LIN {X 0,Y 673.595,Z 978.183,A -85,B 0,C 180,E1 32397.712,E2 32397.712} C_VEL
LIN {X 0,Y 673.691,Z 963.128,A -85,B 0,C 180,E1 32397.38,E2 32397.38} C_VEL
LIN {X 0,Y 673.783,Z 926.963,A -85,B 0,C 180,E1 32396.96,E2 32396.96} C_VEL
LIN {X 0,Y 674.022,Z 820.76,A -85,B 0,C 180,E1 32395.779,E2 32395.779} C_VEL
LIN {X 0,Y 674.488,Z 777.084,A -85,B 0,C 180,E1 32392.62,E2 32392.62} C_VEL
LIN {X 0,Y 674.751,Z 739.413,A -85,B 0,C 180,E1 32389.928,E2 32389.928} C_VEL
LIN {X 0,Y 674.996,Z 702.216,A -85,B 0,C 180,E1 32387.302,E2 32387.302} C_VEL
LIN {X 0,Y 674.853,Z 660.758,A -85,B 0,C 180,E1 32384.443,E2 32384.443} C_VEL
LIN {X 0,Y 674.656,Z 625.3,A -85,B 0,C 180,E1 32382.074,E2 32382.074} C_VEL
LIN {X 0,Y 672.585,Z 616.892,A -85,B 0,C 180,E1 32381.448,E2 32381.448} C_VEL
LIN {X 0,Y 672.585,Z 616.892,A -85,B 0,C 180,E1 32378.297,E2 32378.297} C_VEL
LIN {X 0,Y 672.544,Z 616.896,A -85,B 0,C 180,E1 32375.211,E2 32375.211} C_VEL
LIN {X 0,Y 672.55,Z 616.893,A -85,B 0,C 180,E1 32372.362,E2 32372.362} C_VEL
LIN {X 0,Y 672.577,Z 616.89,A -85,B 0,C 180,E1 32369.233,E2 32369.233} C_VEL
LIN {X 0,Y 672.572,Z 616.892,A -85,B 0,C 180,E1 32366.203,E2 32366.203} C_VEL
LIN {X 0,Y 672.574,Z 616.893,A -85,B 0,C 180,E1 32363.191,E2 32363.191} C_VEL
LIN {X 0,Y 672.566,Z 616.892,A -85,B 0,C 180,E1 32360.227,E2 32360.227} C_VEL
LIN {X 0,Y 672.576,Z 616.888,A -85,B 0,C 180,E1 32357.086,E2 32357.086} C_VEL
LIN {X 0,Y 672.546,Z 616.892,A -85,B 0,C 180,E1 32354.087,E2 32354.087} C_VEL
LIN {X 0,Y 672.591,Z 616.89,A -85,B 0,C 180,E1 32351.076,E2 32351.076} C_VEL
LIN {X 0,Y 672.582,Z 616.891,A -85,B 0,C 180,E1 32347.984,E2 32347.984} C_VEL
LIN {X 0,Y 672.581,Z 616.892,A -85,B 0,C 180,E1 32344.851,E2 32344.851} C_VEL
LIN {X 0,Y 672.566,Z 616.895,A -85,B 0,C 180,E1 32344.293,E2 32344.293} C_VEL
LIN {X 0,Y 678.826,Z 637.109,A -85,B 0,C 180,E1 32342.275,E2 32342.275} C_VEL
LIN {X 0,Y 677.864,Z 671.07,A -85,B 0,C 180,E1 32339.563,E2 32339.563} C_VEL
LIN {X 0,Y 677.664,Z 682.912,A -85,B 0,C 180,E1 32338.655,E2 32338.655} C_VEL
LIN {X 0,Y 681.031,Z 699.716,A -85,B 0,C 180,E1 32338.3,E2 32338.3} C_VEL
LIN {X 0,Y 679.199,Z 978.779,A -85,B 0,C 180,E1 32335.156,E2 32335.156} C_VEL
LIN {X 0,Y 678.886,Z 1000.715,A -85,B 0,C 180,E1 32334.812,E2 32334.812} C_VEL
LIN {X 0,Y 678.362,Z 1022.472,A -85,B 0,C 180,E1 32334.307,E2 32334.307} C_VEL
LIN {X 0,Y 677.771,Z 1043.763,A -85,B 0,C 180,E1 32333.656,E2 32333.656} C_VEL
LIN {X 0,Y 677.123,Z 1063.834,A -85,B 0,C 180,E1 32332.892,E2 32332.892} C_VEL
LIN {X 0,Y 676.435,Z 1082.877,A -85,B 0,C 180,E1 32332.005,E2 32332.005} C_VEL
LIN {X 0,Y 675.676,Z 1102.121,A -85,B 0,C 180,E1 32330.942,E2 32330.942} C_VEL
LIN {X 0,Y 674.981,Z 1120.021,A -85,B 0,C 180,E1 32329.783,E2 32329.783} C_VEL
LIN {X 0,Y 674.308,Z 1136.916,A -85,B 0,C 180,E1 32328.5,E2 32328.5} C_VEL
LIN {X 0,Y 673.686,Z 1152.877,A -85,B 0,C 180,E1 32327.088,E2 32327.088} C_VEL
LIN {X 0,Y 673.175,Z 1167.476,A -85,B 0,C 180,E1 32325.594,E2 32325.594} C_VEL
LIN {X 0,Y 672.763,Z 1180.671,A -85,B 0,C 180,E1 32324.018,E2 32324.018} C_VEL
LIN {X 0,Y 672.436,Z 1192.394,A -85,B 0,C 180,E1 32322.363,E2 32322.363} C_VEL
LIN {X 0,Y 672.2,Z 1203.223,A -85,B 0,C 180,E1 32320.541,E2 32320.541} C_VEL
LIN {X 0,Y 672.056,Z 1211.703,A -85,B 0,C 180,E1 32318.814,E2 32318.814} C_VEL
LIN {X 0,Y 671.961,Z 1218.677,A -85,B 0,C 180,E1 32317.007,E2 32317.007} C_VEL
LIN {X 0,Y 671.917,Z 1224.198,A -85,B 0,C 180,E1 32315.121,E2 32315.121} C_VEL
LIN {X 0,Y 671.906,Z 1227.88,A -85,B 0,C 180,E1 32313.326,E2 32313.326} C_VEL
LIN {X 0,Y 671.901,Z 1229.885,A -85,B 0,C 180,E1 32311.534,E2 32311.534} C_VEL
LIN {X 0,Y 671.899,Z 1230.396,A -85,B 0,C 180,E1 32309.573,E2 32309.573} C_VEL
LIN {X 0,Y 671.913,Z 1229.232,A -85,B 0,C 180,E1 32307.696,E2 32307.696} C_VEL
LIN {X 0,Y 671.922,Z 1226.459,A -85,B 0,C 180,E1 32305.903,E2 32305.903} C_VEL
LIN {X 0,Y 671.934,Z 1221.905,A -85,B 0,C 180,E1 32304.02,E2 32304.02} C_VEL
LIN {X 0,Y 671.99,Z 1215.93,A -85,B 0,C 180,E1 32302.217,E2 32302.217} C_VEL
LIN {X 0,Y 672.093,Z 1208.469,A -85,B 0,C 180,E1 32300.494,E2 32300.494} C_VEL
LIN {X 0,Y 672.279,Z 1198.83,A -85,B 0,C 180,E1 32298.677,E2 32298.677} C_VEL
LIN {X 0,Y 672.551,Z 1188.342,A -85,B 0,C 180,E1 32297.026,E2 32297.026} C_VEL
LIN {X 0,Y 672.903,Z 1175.746,A -85,B 0,C 180,E1 32295.367,E2 32295.367} C_VEL
LIN {X 0,Y 673.372,Z 1161.698,A -85,B 0,C 180,E1 32293.789,E2 32293.789} C_VEL
LIN {X 0,Y 673.953,Z 1146.187,A -85,B 0,C 180,E1 32292.293,E2 32292.293} C_VEL
LIN {X 0,Y 674.602,Z 1129.671,A -85,B 0,C 180,E1 32290.923,E2 32290.923} C_VEL
LIN {X 0,Y 675.282,Z 1112.074,A -85,B 0,C 180,E1 32289.682,E2 32289.682} C_VEL
LIN {X 0,Y 676.046,Z 1092.906,A -85,B 0,C 180,E1 32288.526,E2 32288.526} C_VEL
LIN {X 0,Y 676.778,Z 1073.721,A -85,B 0,C 180,E1 32287.547,E2 32287.547} C_VEL
LIN {X 0,Y 677.469,Z 1053.6,A -85,B 0,C 180,E1 32286.699,E2 32286.699} C_VEL
LIN {X 0,Y 678.09,Z 1032.642,A -85,B 0,C 180,E1 32285.984,E2 32285.984} C_VEL
LIN {X 0,Y 678.646,Z 1011.301,A -85,B 0,C 180,E1 32285.414,E2 32285.414} C_VEL
LIN {X 0,Y 679.058,Z 989.931,A -85,B 0,C 180,E1 32285,E2 32285} C_VEL
LIN {X 0,Y 679.387,Z 956.893,A -85,B 0,C 180,E1 32284.593,E2 32284.593} C_VEL
LIN {X 0,Y 680.928,Z 698.596,A -85,B 0,C 180,E1 32281.704,E2 32281.704} C_VEL
LIN {X 0,Y 677.358,Z 681.383,A -85,B 0,C 180,E1 32281.33,E2 32281.33} C_VEL
LIN {X 0,Y 678.154,Z 642.731,A -85,B 0,C 180,E1 32278.338,E2 32278.338} C_VEL
LIN {X 0,Y 678.247,Z 636.016,A -85,B 0,C 180,E1 32277.803,E2 32277.803} C_VEL
LIN {X 0,Y 672.566,Z 616.894,A -85,B 0,C 180,E1 32275.91,E2 32275.91} C_VEL
LIN {X 0,Y 672.583,Z 616.889,A -85,B 0,C 180,E1 32272.831,E2 32272.831} C_VEL
LIN {X 0,Y 672.559,Z 616.894,A -85,B 0,C 180,E1 32269.817,E2 32269.817} C_VEL
LIN {X 0,Y 672.579,Z 616.886,A -85,B 0,C 180,E1 32266.853,E2 32266.853} C_VEL
LIN {X 0,Y 672.553,Z 616.894,A -85,B 0,C 180,E1 32263.735,E2 32263.735} C_VEL
LIN {X 0,Y 672.566,Z 616.888,A -85,B 0,C 180,E1 32260.824,E2 32260.824} C_VEL
LIN {X 0,Y 672.548,Z 616.894,A -85,B 0,C 180,E1 32257.666,E2 32257.666} C_VEL
LIN {X 0,Y 672.546,Z 616.891,A -85,B 0,C 180,E1 32254.814,E2 32254.814} C_VEL
LIN {X 0,Y 672.548,Z 616.896,A -85,B 0,C 180,E1 32251.657,E2 32251.657} C_VEL
LIN {X 0,Y 672.584,Z 617.001,A -85,B 0,C 180,E1 32249.822,E2 32249.822} C_VEL
LIN {X 0,Y 675.411,Z 626.556,A -85,B 0,C 180,E1 32248.699,E2 32248.699} C_VEL
LIN {X 0,Y 680.163,Z 637.227,A -85,B 0,C 180,E1 32248.344,E2 32248.344} C_VEL
LIN {X 0,Y 681.085,Z 642.185,A -85,B 0,C 180,E1 32248.239,E2 32248.239} C_VEL
LIN {X 0,Y 680.031,Z 786.399,A -85,B 0,C 180,E1 32246.589,E2 32246.589} C_VEL
LIN {X 0,Y 679.147,Z 925.853,A -85,B 0,C 180,E1 32245.017,E2 32245.017} C_VEL
LIN {X 0,Y 678.707,Z 947.734,A -85,B 0,C 180,E1 32244.618,E2 32244.618} C_VEL
LIN {X 0,Y 678.186,Z 969.69,A -85,B 0,C 180,E1 32244.059,E2 32244.059} C_VEL
LIN {X 0,Y 677.577,Z 990.34,A -85,B 0,C 180,E1 32243.382,E2 32243.382} C_VEL
LIN {X 0,Y 676.878,Z 1010.769,A -85,B 0,C 180,E1 32242.542,E2 32242.542} C_VEL
LIN {X 0,Y 676.134,Z 1030.476,A -85,B 0,C 180,E1 32241.562,E2 32241.562} C_VEL
LIN {X 0,Y 675.378,Z 1049.81,A -85,B 0,C 180,E1 32240.421,E2 32240.421} C_VEL
LIN {X 0,Y 674.676,Z 1067.906,A -85,B 0,C 180,E1 32239.165,E2 32239.165} C_VEL
LIN {X 0,Y 673.985,Z 1085.338,A -85,B 0,C 180,E1 32237.741,E2 32237.741} C_VEL
LIN {X 0,Y 673.419,Z 1100.427,A -85,B 0,C 180,E1 32236.299,E2 32236.299} C_VEL
LIN {X 0,Y 672.932,Z 1114.879,A -85,B 0,C 180,E1 32234.692,E2 32234.692} C_VEL
LIN {X 0,Y 672.571,Z 1127.414,A -85,B 0,C 180,E1 32233.062,E2 32233.062} C_VEL
LIN {X 0,Y 672.289,Z 1138.579,A -85,B 0,C 180,E1 32231.324,E2 32231.324} C_VEL
LIN {X 0,Y 672.109,Z 1148.379,A -85,B 0,C 180,E1 32229.48,E2 32229.48} C_VEL
LIN {X 0,Y 672.001,Z 1156.064,A -85,B 0,C 180,E1 32227.697,E2 32227.697} C_VEL
LIN {X 0,Y 671.931,Z 1162.036,A -85,B 0,C 180,E1 32225.895,E2 32225.895} C_VEL
LIN {X 0,Y 671.906,Z 1166.534,A -85,B 0,C 180,E1 32224.012,E2 32224.012} C_VEL
LIN {X 0,Y 671.899,Z 1169.286,A -85,B 0,C 180,E1 32222.219,E2 32222.219} C_VEL
LIN {X 0,Y 671.899,Z 1170.383,A -85,B 0,C 180,E1 32220.428,E2 32220.428} C_VEL
LIN {X 0,Y 671.904,Z 1169.924,A -85,B 0,C 180,E1 32218.467,E2 32218.467} C_VEL
LIN {X 0,Y 671.917,Z 1167.817,A -85,B 0,C 180,E1 32216.589,E2 32216.589} C_VEL
LIN {X 0,Y 671.936,Z 1163.894,A -85,B 0,C 180,E1 32214.708,E2 32214.708} C_VEL
LIN {X 0,Y 671.976,Z 1158.25,A -85,B 0,C 180,E1 32212.822,E2 32212.822} C_VEL
LIN {X 0,Y 672.069,Z 1151.145,A -85,B 0,C 180,E1 32211.015,E2 32211.015} C_VEL
LIN {X 0,Y 672.209,Z 1142.536,A -85,B 0,C 180,E1 32209.287,E2 32209.287} C_VEL
LIN {X 0,Y 672.457,Z 1131.561,A -85,B 0,C 180,E1 32207.464,E2 32207.464} C_VEL
LIN {X 0,Y 672.797,Z 1119.676,A -85,B 0,C 180,E1 32205.808,E2 32205.808} C_VEL
LIN {X 0,Y 673.217,Z 1106.283,A -85,B 0,C 180,E1 32204.231,E2 32204.231} C_VEL
LIN {X 0,Y 673.737,Z 1091.522,A -85,B 0,C 180,E1 32202.736,E2 32202.736} C_VEL
LIN {X 0,Y 674.39,Z 1074.768,A -85,B 0,C 180,E1 32201.279,E2 32201.279} C_VEL
LIN {X 0,Y 675.116,Z 1056.843,A -85,B 0,C 180,E1 32199.951,E2 32199.951} C_VEL
LIN {X 0,Y 675.826,Z 1038.474,A -85,B 0,C 180,E1 32198.795,E2 32198.795} C_VEL
LIN {X 0,Y 676.56,Z 1019.286,A -85,B 0,C 180,E1 32197.771,E2 32197.771} C_VEL
LIN {X 0,Y 677.275,Z 999.369,A -85,B 0,C 180,E1 32196.879,E2 32196.879} C_VEL
LIN {X 0,Y 677.954,Z 978.015,A -85,B 0,C 180,E1 32196.102,E2 32196.102} C_VEL
LIN {X 0,Y 678.522,Z 956.689,A -85,B 0,C 180,E1 32195.5,E2 32195.5} C_VEL
LIN {X 0,Y 678.953,Z 934.57,A -85,B 0,C 180,E1 32195.034,E2 32195.034} C_VEL
LIN {X 0,Y 678.228,Z 927.061,A -85,B 0,C 180,E1 32194.873,E2 32194.873} C_VEL
LIN {X 0,Y 672.708,Z 907.3,A -85,B 0,C 180,E1 32194.41,E2 32194.41} C_VEL
LIN {X 0,Y 672.056,Z 900.783,A -85,B 0,C 180,E1 32194.312,E2 32194.312} C_VEL
LIN {X 0,Y 673.767,Z 674.641,A -85,B 0,C 180,E1 32191.732,E2 32191.732} C_VEL
LIN {X 0,Y 673.889,Z 642.039,A -85,B 0,C 180,E1 32191.338,E2 32191.338} C_VEL
LIN {X 0,Y 672.187,Z 636.898,A -85,B 0,C 180,E1 32191.193,E2 32191.193} C_VEL
LIN {X 0,Y 666.544,Z 624.913,A -85,B 0,C 180,E1 32190.763,E2 32190.763} C_VEL
LIN {X 0,Y 664.595,Z 617.887,A -85,B 0,C 180,E1 32189.937,E2 32189.937} C_VEL
LIN {X 0,Y 664.571,Z 617.887,A -85,B 0,C 180,E1 32187.252,E2 32187.252} C_VEL
LIN {X 0,Y 664.597,Z 617.88,A -85,B 0,C 180,E1 32184.04,E2 32184.04} C_VEL
LIN {X 0,Y 664.643,Z 617.881,A -85,B 0,C 180,E1 32181.15,E2 32181.15} C_VEL
LIN {X 0,Y 664.634,Z 617.874,A -85,B 0,C 180,E1 32178.004,E2 32178.004} C_VEL
LIN {X 0,Y 664.613,Z 617.879,A -85,B 0,C 180,E1 32175.122,E2 32175.122} C_VEL
LIN {X 0,Y 664.647,Z 617.878,A -85,B 0,C 180,E1 32172.131,E2 32172.131} C_VEL
LIN {X 0,Y 664.561,Z 617.883,A -85,B 0,C 180,E1 32169.193,E2 32169.193} C_VEL
LIN {X 0,Y 664.641,Z 617.882,A -85,B 0,C 180,E1 32166.352,E2 32166.352} C_VEL
LIN {X 0,Y 664.61,Z 617.877,A -85,B 0,C 180,E1 32163.308,E2 32163.308} C_VEL
LIN {X 0,Y 664.633,Z 617.876,A -85,B 0,C 180,E1 32160.364,E2 32160.364} C_VEL
LIN {X 0,Y 664.648,Z 617.879,A -85,B 0,C 180,E1 32157.313,E2 32157.313} C_VEL
LIN {X 0,Y 664.585,Z 617.881,A -85,B 0,C 180,E1 32154.441,E2 32154.441} C_VEL
LIN {X 0,Y 664.637,Z 617.881,A -85,B 0,C 180,E1 32151.536,E2 32151.536} C_VEL
LIN {X 0,Y 664.578,Z 617.88,A -85,B 0,C 180,E1 32148.592,E2 32148.592} C_VEL
LIN {X 0,Y 664.648,Z 617.874,A -85,B 0,C 180,E1 32145.623,E2 32145.623} C_VEL
LIN {X 0,Y 664.633,Z 617.875,A -85,B 0,C 180,E1 32142.601,E2 32142.601} C_VEL
LIN {X 0,Y 664.62,Z 617.874,A -85,B 0,C 180,E1 32139.614,E2 32139.614} C_VEL
LIN {X 0,Y 664.605,Z 617.882,A -85,B 0,C 180,E1 32136.48,E2 32136.48} C_VEL
LIN {X 0,Y 664.565,Z 617.881,A -85,B 0,C 180,E1 32133.797,E2 32133.797} C_VEL
LIN {X 0,Y 664.597,Z 617.878,A -85,B 0,C 180,E1 32130.605,E2 32130.605} C_VEL
LIN {X 0,Y 664.627,Z 617.88,A -85,B 0,C 180,E1 32127.76,E2 32127.76} C_VEL
LIN {X 0,Y 664.637,Z 617.87,A -85,B 0,C 180,E1 32124.649,E2 32124.649} C_VEL
LIN {X 0,Y 664.615,Z 617.878,A -85,B 0,C 180,E1 32121.61,E2 32121.61} C_VEL
LIN {X 0,Y 664.647,Z 617.871,A -85,B 0,C 180,E1 32118.635,E2 32118.635} C_VEL
LIN {X 0,Y 664.559,Z 617.882,A -85,B 0,C 180,E1 32115.674,E2 32115.674} C_VEL
LIN {X 0,Y 664.644,Z 617.88,A -85,B 0,C 180,E1 32112.792,E2 32112.792} C_VEL
LIN {X 0,Y 664.606,Z 617.877,A -85,B 0,C 180,E1 32109.757,E2 32109.757} C_VEL
LIN {X 0,Y 664.633,Z 617.875,A -85,B 0,C 180,E1 32106.802,E2 32106.802} C_VEL
LIN {X 0,Y 664.645,Z 617.879,A -85,B 0,C 180,E1 32103.71,E2 32103.71} C_VEL
LIN {X 0,Y 664.588,Z 617.879,A -85,B 0,C 180,E1 32100.828,E2 32100.828} C_VEL
LIN {X 0,Y 664.611,Z 617.883,A -85,B 0,C 180,E1 32097.822,E2 32097.822} C_VEL
LIN {X 0,Y 664.577,Z 617.882,A -85,B 0,C 180,E1 32095.026,E2 32095.026} C_VEL
LIN {X 0,Y 664.651,Z 617.874,A -85,B 0,C 180,E1 32092.022,E2 32092.022} C_VEL
LIN {X 0,Y 664.647,Z 617.88,A -85,B 0,C 180,E1 32088.899,E2 32088.899} C_VEL
LIN {X 0,Y 664.649,Z 617.873,A -85,B 0,C 180,E1 32085.729,E2 32085.729} C_VEL
LIN {X 0,Y 664.589,Z 617.883,A -85,B 0,C 180,E1 32082.726,E2 32082.726} C_VEL
LIN {X 0,Y 664.586,Z 617.886,A -85,B 0,C 180,E1 32080.024,E2 32080.024} C_VEL
LIN {X 0,Y 664.607,Z 618.001,A -85,B 0,C 180,E1 32079.231,E2 32079.231} C_VEL
LIN {X 0,Y 668.154,Z 632.235,A -85,B 0,C 180,E1 32078.062,E2 32078.062} C_VEL
LIN {X 0,Y 667.749,Z 675.946,A -85,B 0,C 180,E1 32074.861,E2 32074.861} C_VEL
LIN {X 0,Y 667.355,Z 714.917,A -85,B 0,C 180,E1 32072.006,E2 32072.006} C_VEL
LIN {X 0,Y 666.88,Z 756.424,A -85,B 0,C 180,E1 32068.963,E2 32068.963} C_VEL
LIN {X 0,Y 666.283,Z 796.959,A -85,B 0,C 180,E1 32065.987,E2 32065.987} C_VEL
LIN {X 0,Y 666.079,Z 820.132,A -85,B 0,C 180,E1 32064.313,E2 32064.313} C_VEL
LIN {X 0,Y 666.466,Z 828.042,A -85,B 0,C 180,E1 32064.214,E2 32064.214} C_VEL
LIN {X 0,Y 665.888,Z 961.771,A -85,B 0,C 180,E1 32062.703,E2 32062.703} C_VEL
LIN {X 0,Y 665.772,Z 977.873,A -85,B 0,C 180,E1 32062.361,E2 32062.361} C_VEL
LIN {X 0,Y 665.603,Z 994.084,A -85,B 0,C 180,E1 32061.845,E2 32061.845} C_VEL
LIN {X 0,Y 665.386,Z 1008.252,A -85,B 0,C 180,E1 32061.23,E2 32061.23} C_VEL
LIN {X 0,Y 665.159,Z 1022.895,A -85,B 0,C 180,E1 32060.408,E2 32060.408} C_VEL
LIN {X 0,Y 664.906,Z 1035.605,A -85,B 0,C 180,E1 32059.5,E2 32059.5} C_VEL
LIN {X 0,Y 664.689,Z 1046.829,A -85,B 0,C 180,E1 32058.504,E2 32058.504} C_VEL
LIN {X 0,Y 664.497,Z 1056.655,A -85,B 0,C 180,E1 32057.422,E2 32057.422} C_VEL
LIN {X 0,Y 664.338,Z 1065.659,A -85,B 0,C 180,E1 32056.165,E2 32056.165} C_VEL
LIN {X 0,Y 664.233,Z 1072.65,A -85,B 0,C 180,E1 32054.898,E2 32054.898} C_VEL
LIN {X 0,Y 664.173,Z 1078.359,A -85,B 0,C 180,E1 32053.47,E2 32053.47} C_VEL
LIN {X 0,Y 664.13,Z 1082.281,A -85,B 0,C 180,E1 32051.901,E2 32051.901} C_VEL
LIN {X 0,Y 664.117,Z 1083.917,A -85,B 0,C 180,E1 32050.494,E2 32050.494} C_VEL
LIN {X 0,Y 664.134,Z 1083.67,A -85,B 0,C 180,E1 32049.006,E2 32049.006} C_VEL
LIN {X 0,Y 664.159,Z 1081.674,A -85,B 0,C 180,E1 32047.611,E2 32047.611} C_VEL
LIN {X 0,Y 664.203,Z 1077.548,A -85,B 0,C 180,E1 32046.134,E2 32046.134} C_VEL
LIN {X 0,Y 664.287,Z 1072.092,A -85,B 0,C 180,E1 32044.833,E2 32044.833} C_VEL
LIN {X 0,Y 664.407,Z 1064.701,A -85,B 0,C 180,E1 32043.536,E2 32043.536} C_VEL
LIN {X 0,Y 664.562,Z 1056.501,A -85,B 0,C 180,E1 32042.413,E2 32042.413} C_VEL
LIN {X 0,Y 664.768,Z 1046.138,A -85,B 0,C 180,E1 32041.291,E2 32041.291} C_VEL
LIN {X 0,Y 665.002,Z 1034.772,A -85,B 0,C 180,E1 32040.3,E2 32040.3} C_VEL
LIN {X 0,Y 665.234,Z 1021.705,A -85,B 0,C 180,E1 32039.395,E2 32039.395} C_VEL
LIN {X 0,Y 665.432,Z 1007.588,A -85,B 0,C 180,E1 32038.621,E2 32038.621} C_VEL
LIN {X 0,Y 665.633,Z 993.046,A -85,B 0,C 180,E1 32038.018,E2 32038.018} C_VEL
LIN {X 0,Y 665.772,Z 979.228,A -85,B 0,C 180,E1 32037.588,E2 32037.588} C_VEL
LIN {X 0,Y 665.863,Z 964.186,A -85,B 0,C 180,E1 32037.252,E2 32037.252} C_VEL
LIN {X 0,Y 665.972,Z 925.839,A -85,B 0,C 180,E1 32036.8,E2 32036.8} C_VEL
LIN {X 0,Y 666.29,Z 821.623,A -85,B 0,C 180,E1 32035.614,E2 32035.614} C_VEL
LIN {X 0,Y 666.775,Z 779.969,A -85,B 0,C 180,E1 32032.589,E2 32032.589} C_VEL
LIN {X 0,Y 667.072,Z 741.938,A -85,B 0,C 180,E1 32029.854,E2 32029.854} C_VEL
LIN {X 0,Y 667.309,Z 704.066,A -85,B 0,C 180,E1 32027.186,E2 32027.186} C_VEL
LIN {X 0,Y 667.227,Z 666.344,A -85,B 0,C 180,E1 32024.572,E2 32024.572} C_VEL
LIN {X 0,Y 667.088,Z 627.617,A -85,B 0,C 180,E1 32021.968,E2 32021.968} C_VEL
LIN {X 0,Y 664.64,Z 617.882,A -85,B 0,C 180,E1 32021.241,E2 32021.241} C_VEL
LIN {X 0,Y 664.647,Z 617.879,A -85,B 0,C 180,E1 32018.092,E2 32018.092} C_VEL
LIN {X 0,Y 664.606,Z 617.885,A -85,B 0,C 180,E1 32014.894,E2 32014.894} C_VEL
LIN {X 0,Y 664.632,Z 617.881,A -85,B 0,C 180,E1 32011.907,E2 32011.907} C_VEL
LIN {X 0,Y 664.645,Z 617.881,A -85,B 0,C 180,E1 32008.833,E2 32008.833} C_VEL
LIN {X 0,Y 664.65,Z 617.877,A -85,B 0,C 180,E1 32005.677,E2 32005.677} C_VEL
LIN {X 0,Y 664.604,Z 617.882,A -85,B 0,C 180,E1 32002.567,E2 32002.567} C_VEL
LIN {X 0,Y 664.635,Z 617.879,A -85,B 0,C 180,E1 31999.577,E2 31999.577} C_VEL
LIN {X 0,Y 664.642,Z 617.879,A -85,B 0,C 180,E1 31996.446,E2 31996.446} C_VEL
LIN {X 0,Y 664.65,Z 617.877,A -85,B 0,C 180,E1 31993.312,E2 31993.312} C_VEL
LIN {X 0,Y 664.603,Z 617.883,A -85,B 0,C 180,E1 31990.195,E2 31990.195} C_VEL
LIN {X 0,Y 664.637,Z 617.877,A -85,B 0,C 180,E1 31987.21,E2 31987.21} C_VEL
LIN {X 0,Y 664.639,Z 617.944,A -85,B 0,C 180,E1 31984.645,E2 31984.645} C_VEL
LIN {X 0,Y 671.478,Z 640.085,A -85,B 0,C 180,E1 31982.4,E2 31982.4} C_VEL
LIN {X 0,Y 670.318,Z 675.625,A -85,B 0,C 180,E1 31979.536,E2 31979.536} C_VEL
LIN {X 0,Y 670.218,Z 682.595,A -85,B 0,C 180,E1 31979.003,E2 31979.003} C_VEL
LIN {X 0,Y 673.916,Z 701.089,A -85,B 0,C 180,E1 31978.597,E2 31978.597} C_VEL
LIN {X 0,Y 672.129,Z 947.209,A -85,B 0,C 180,E1 31975.791,E2 31975.791} C_VEL
LIN {X 0,Y 671.745,Z 988.99,A -85,B 0,C 180,E1 31975.288,E2 31975.288} C_VEL
LIN {X 0,Y 671.3,Z 1010.943,A -85,B 0,C 180,E1 31974.869,E2 31974.869} C_VEL
LIN {X 0,Y 670.765,Z 1031.934,A -85,B 0,C 180,E1 31974.316,E2 31974.316} C_VEL
LIN {X 0,Y 670.107,Z 1052.298,A -85,B 0,C 180,E1 31973.626,E2 31973.626} C_VEL
LIN {X 0,Y 669.376,Z 1071.765,A -85,B 0,C 180,E1 31972.806,E2 31972.806} C_VEL
LIN {X 0,Y 668.556,Z 1091.32,A -85,B 0,C 180,E1 31971.816,E2 31971.816} C_VEL
LIN {X 0,Y 667.76,Z 1110.103,A -85,B 0,C 180,E1 31970.693,E2 31970.693} C_VEL
LIN {X 0,Y 666.979,Z 1127.926,A -85,B 0,C 180,E1 31969.438,E2 31969.438} C_VEL
LIN {X 0,Y 666.256,Z 1144.186,A -85,B 0,C 180,E1 31968.097,E2 31968.097} C_VEL
LIN {X 0,Y 665.604,Z 1160.076,A -85,B 0,C 180,E1 31966.578,E2 31966.578} C_VEL
LIN {X 0,Y 665.115,Z 1173.638,A -85,B 0,C 180,E1 31965.073,E2 31965.073} C_VEL
LIN {X 0,Y 664.692,Z 1185.823,A -85,B 0,C 180,E1 31963.482,E2 31963.482} C_VEL
LIN {X 0,Y 664.368,Z 1197.301,A -85,B 0,C 180,E1 31961.721,E2 31961.721} C_VEL
LIN {X 0,Y 664.159,Z 1206.858,A -85,B 0,C 180,E1 31959.969,E2 31959.969} C_VEL
LIN {X 0,Y 664.034,Z 1214.53,A -85,B 0,C 180,E1 31958.223,E2 31958.223} C_VEL
LIN {X 0,Y 663.954,Z 1221.158,A -85,B 0,C 180,E1 31956.308,E2 31956.308} C_VEL
LIN {X 0,Y 663.927,Z 1225.919,A -85,B 0,C 180,E1 31954.44,E2 31954.44} C_VEL
LIN {X 0,Y 663.914,Z 1228.902,A -85,B 0,C 180,E1 31952.588,E2 31952.588} C_VEL
LIN {X 0,Y 663.905,Z 1230.328,A -85,B 0,C 180,E1 31950.689,E2 31950.689} C_VEL
LIN {X 0,Y 663.903,Z 1230.208,A -85,B 0,C 180,E1 31948.877,E2 31948.877} C_VEL
LIN {X 0,Y 663.905,Z 1228.444,A -85,B 0,C 180,E1 31947.064,E2 31947.064} C_VEL
LIN {X 0,Y 663.912,Z 1225.013,A -85,B 0,C 180,E1 31945.161,E2 31945.161} C_VEL
LIN {X 0,Y 663.954,Z 1220.127,A -85,B 0,C 180,E1 31943.34,E2 31943.34} C_VEL
LIN {X 0,Y 664.049,Z 1213.46,A -85,B 0,C 180,E1 31941.513,E2 31941.513} C_VEL
LIN {X 0,Y 664.19,Z 1205.042,A -85,B 0,C 180,E1 31939.679,E2 31939.679} C_VEL
LIN {X 0,Y 664.42,Z 1195.218,A -85,B 0,C 180,E1 31937.925,E2 31937.925} C_VEL
LIN {X 0,Y 664.745,Z 1183.902,A -85,B 0,C 180,E1 31936.251,E2 31936.251} C_VEL
LIN {X 0,Y 665.215,Z 1170.538,A -85,B 0,C 180,E1 31934.57,E2 31934.57} C_VEL
LIN {X 0,Y 665.764,Z 1156.557,A -85,B 0,C 180,E1 31933.06,E2 31933.06} C_VEL
LIN {X 0,Y 666.415,Z 1140.789,A -85,B 0,C 180,E1 31931.604,E2 31931.604} C_VEL
LIN {X 0,Y 667.133,Z 1123.86,A -85,B 0,C 180,E1 31930.262,E2 31930.262} C_VEL
LIN {X 0,Y 667.944,Z 1105.826,A -85,B 0,C 180,E1 31929.035,E2 31929.035} C_VEL
LIN {X 0,Y 668.749,Z 1087.225,A -85,B 0,C 180,E1 31927.957,E2 31927.957} C_VEL
LIN {X 0,Y 669.525,Z 1067.695,A -85,B 0,C 180,E1 31927.012,E2 31927.012} C_VEL
LIN {X 0,Y 670.31,Z 1046.263,A -85,B 0,C 180,E1 31926.155,E2 31926.155} C_VEL
LIN {X 0,Y 670.94,Z 1026.608,A -85,B 0,C 180,E1 31925.524,E2 31925.524} C_VEL
LIN {X 0,Y 671.388,Z 1005.306,A -85,B 0,C 180,E1 31925.017,E2 31925.017} C_VEL
LIN {X 0,Y 671.767,Z 981.923,A -85,B 0,C 180,E1 31924.625,E2 31924.625} C_VEL
LIN {X 0,Y 673.307,Z 755.89,A -85,B 0,C 180,E1 31922.072,E2 31922.072} C_VEL
LIN {X 0,Y 673.604,Z 699.079,A -85,B 0,C 180,E1 31921.39,E2 31921.39} C_VEL
LIN {X 0,Y 669.798,Z 680.518,A -85,B 0,C 180,E1 31920.976,E2 31920.976} C_VEL
LIN {X 0,Y 670.742,Z 643.003,A -85,B 0,C 180,E1 31918.02,E2 31918.02} C_VEL
LIN {X 0,Y 670.723,Z 638.399,A -85,B 0,C 180,E1 31917.643,E2 31917.643} C_VEL
LIN {X 0,Y 664.94,Z 619.335,A -85,B 0,C 180,E1 31915.722,E2 31915.722} C_VEL
LIN {X 0,Y 664.62,Z 617.883,A -85,B 0,C 180,E1 31915.55,E2 31915.55} C_VEL
LIN {X 0,Y 664.64,Z 617.88,A -85,B 0,C 180,E1 31912.57,E2 31912.57} C_VEL
LIN {X 0,Y 664.615,Z 617.882,A -85,B 0,C 180,E1 31909.69,E2 31909.69} C_VEL
LIN {X 0,Y 664.646,Z 617.877,A -85,B 0,C 180,E1 31906.685,E2 31906.685} C_VEL
LIN {X 0,Y 664.611,Z 617.883,A -85,B 0,C 180,E1 31903.643,E2 31903.643} C_VEL
LIN {X 0,Y 664.644,Z 617.877,A -85,B 0,C 180,E1 31900.649,E2 31900.649} C_VEL
LIN {X 0,Y 664.6,Z 617.883,A -85,B 0,C 180,E1 31897.542,E2 31897.542} C_VEL
LIN {X 0,Y 664.622,Z 617.879,A -85,B 0,C 180,E1 31894.66,E2 31894.66} C_VEL
LIN {X 0,Y 664.601,Z 617.886,A -85,B 0,C 180,E1 31891.573,E2 31891.573} C_VEL
LIN {X 0,Y 664.673,Z 618.025,A -85,B 0,C 180,E1 31890.213,E2 31890.213} C_VEL
LIN {X 0,Y 667.482,Z 627.482,A -85,B 0,C 180,E1 31889.063,E2 31889.063} C_VEL
LIN {X 0,Y 673.413,Z 639.997,A -85,B 0,C 180,E1 31888.621,E2 31888.621} C_VEL
LIN {X 0,Y 674.03,Z 643.813,A -85,B 0,C 180,E1 31888.544,E2 31888.544} C_VEL
LIN {X 0,Y 672.696,Z 785.858,A -85,B 0,C 180,E1 31886.866,E2 31886.866} C_VEL
LIN {X 0,Y 671.762,Z 927.523,A -85,B 0,C 180,E1 31885.261,E2 31885.261} C_VEL
LIN {X 0,Y 671.318,Z 949.818,A -85,B 0,C 180,E1 31884.847,E2 31884.847} C_VEL
LIN {X 0,Y 670.793,Z 971.156,A -85,B 0,C 180,E1 31884.295,E2 31884.295} C_VEL
LIN {X 0,Y 670.158,Z 990.826,A -85,B 0,C 180,E1 31883.637,E2 31883.637} C_VEL
LIN {X 0,Y 669.414,Z 1010.673,A -85,B 0,C 180,E1 31882.812,E2 31882.812} C_VEL
LIN {X 0,Y 668.593,Z 1030.479,A -85,B 0,C 180,E1 31881.818,E2 31881.818} C_VEL
LIN {X 0,Y 667.789,Z 1049.351,A -85,B 0,C 180,E1 31880.695,E2 31880.695} C_VEL
LIN {X 0,Y 667.012,Z 1067.334,A -85,B 0,C 180,E1 31879.44,E2 31879.44} C_VEL
LIN {X 0,Y 666.242,Z 1084.723,A -85,B 0,C 180,E1 31878.01,E2 31878.01} C_VEL
LIN {X 0,Y 665.596,Z 1100.428,A -85,B 0,C 180,E1 31876.496,E2 31876.496} C_VEL
LIN {X 0,Y 665.064,Z 1114.642,A -85,B 0,C 180,E1 31874.899,E2 31874.899} C_VEL
LIN {X 0,Y 664.655,Z 1127.418,A -85,B 0,C 180,E1 31873.22,E2 31873.22} C_VEL
LIN {X 0,Y 664.339,Z 1138.584,A -85,B 0,C 180,E1 31871.461,E2 31871.461} C_VEL
LIN {X 0,Y 664.135,Z 1148.254,A -85,B 0,C 180,E1 31869.622,E2 31869.622} C_VEL
LIN {X 0,Y 664.009,Z 1156.064,A -85,B 0,C 180,E1 31867.791,E2 31867.791} C_VEL
LIN {X 0,Y 663.936,Z 1162.039,A -85,B 0,C 180,E1 31865.966,E2 31865.966} C_VEL
LIN {X 0,Y 663.907,Z 1166.533,A -85,B 0,C 180,E1 31864.061,E2 31864.061} C_VEL
LIN {X 0,Y 663.9,Z 1169.286,A -85,B 0,C 180,E1 31862.246,E2 31862.246} C_VEL
LIN {X 0,Y 663.899,Z 1170.383,A -85,B 0,C 180,E1 31860.433,E2 31860.433} C_VEL
LIN {X 0,Y 663.904,Z 1169.924,A -85,B 0,C 180,E1 31858.448,E2 31858.448} C_VEL
LIN {X 0,Y 663.917,Z 1167.815,A -85,B 0,C 180,E1 31856.548,E2 31856.548} C_VEL
LIN {X 0,Y 663.937,Z 1164.101,A -85,B 0,C 180,E1 31854.731,E2 31854.731} C_VEL
LIN {X 0,Y 663.98,Z 1158.552,A -85,B 0,C 180,E1 31852.822,E2 31852.822} C_VEL
LIN {X 0,Y 664.081,Z 1151.506,A -85,B 0,C 180,E1 31850.993,E2 31850.993} C_VEL
LIN {X 0,Y 664.236,Z 1142.999,A -85,B 0,C 180,E1 31849.244,E2 31849.244} C_VEL
LIN {X 0,Y 664.495,Z 1132.719,A -85,B 0,C 180,E1 31847.488,E2 31847.488} C_VEL
LIN {X 0,Y 664.855,Z 1121.001,A -85,B 0,C 180,E1 31845.812,E2 31845.812} C_VEL
LIN {X 0,Y 665.31,Z 1107.854,A -85,B 0,C 180,E1 31844.218,E2 31844.218} C_VEL
LIN {X 0,Y 665.879,Z 1093.411,A -85,B 0,C 180,E1 31842.706,E2 31842.706} C_VEL
LIN {X 0,Y 666.585,Z 1076.974,A -85,B 0,C 180,E1 31841.233,E2 31841.233} C_VEL
LIN {X 0,Y 667.353,Z 1059.348,A -85,B 0,C 180,E1 31839.89,E2 31839.89} C_VEL
LIN {X 0,Y 668.154,Z 1040.704,A -85,B 0,C 180,E1 31838.678,E2 31838.678} C_VEL
LIN {X 0,Y 668.996,Z 1021.097,A -85,B 0,C 180,E1 31837.599,E2 31837.599} C_VEL
LIN {X 0,Y 669.796,Z 1000.944,A -85,B 0,C 180,E1 31836.671,E2 31836.671} C_VEL
LIN {X 0,Y 670.525,Z 979.828,A -85,B 0,C 180,E1 31835.886,E2 31835.886} C_VEL
LIN {X 0,Y 671.13,Z 958.705,A -85,B 0,C 180,E1 31835.273,E2 31835.273} C_VEL
LIN {X 0,Y 671.609,Z 936.489,A -85,B 0,C 180,E1 31834.79,E2 31834.79} C_VEL
LIN {X 0,Y 671.957,Z 913.789,A -85,B 0,C 180,E1 31834.46,E2 31834.46} C_VEL
LIN {X 0,Y 672.056,Z 900.783,A -85,B 0,C 180,E1 31834.312,E2 31834.312} C_VEL
LIN {X 0,Y 671.193,Z 893.193,A -85,B 0,C 180,E1 31834.192,E2 31834.192} C_VEL
LIN {X 0,Y 665.618,Z 873.352,A -85,B 0,C 180,E1 31833.748,E2 31833.748} C_VEL
LIN {X 0,Y 664.985,Z 866.827,A -85,B 0,C 180,E1 31833.647,E2 31833.647} C_VEL
LIN {X 0,Y 666.945,Z 652.013,A -85,B 0,C 180,E1 31831.14,E2 31831.14} C_VEL
LIN {X 0,Y 666.846,Z 643.607,A -85,B 0,C 180,E1 31831.026,E2 31831.026} C_VEL
LIN {X 0,Y 662.12,Z 632.926,A -85,B 0,C 180,E1 31830.66,E2 31830.66} C_VEL
LIN {X 0,Y 658.499,Z 625.29,A -85,B 0,C 180,E1 31830.379,E2 31830.379} C_VEL
LIN {X 0,Y 656.638,Z 618.878,A -85,B 0,C 180,E1 31829.61,E2 31829.61} C_VEL
LIN {X 0,Y 656.694,Z 618.872,A -85,B 0,C 180,E1 31826.659,E2 31826.659} C_VEL
LIN {X 0,Y 656.649,Z 618.87,A -85,B 0,C 180,E1 31823.661,E2 31823.661} C_VEL
LIN {X 0,Y 656.706,Z 618.863,A -85,B 0,C 180,E1 31820.702,E2 31820.702} C_VEL
LIN {X 0,Y 656.702,Z 618.867,A -85,B 0,C 180,E1 31817.588,E2 31817.588} C_VEL
LIN {X 0,Y 656.68,Z 618.864,A -85,B 0,C 180,E1 31814.557,E2 31814.557} C_VEL
LIN {X 0,Y 656.646,Z 618.872,A -85,B 0,C 180,E1 31811.366,E2 31811.366} C_VEL
LIN {X 0,Y 656.643,Z 618.872,A -85,B 0,C 180,E1 31808.633,E2 31808.633} C_VEL
LIN {X 0,Y 656.664,Z 618.865,A -85,B 0,C 180,E1 31805.568,E2 31805.568} C_VEL
LIN {X 0,Y 656.706,Z 618.868,A -85,B 0,C 180,E1 31802.616,E2 31802.616} C_VEL
LIN {X 0,Y 656.702,Z 618.862,A -85,B 0,C 180,E1 31799.56,E2 31799.56} C_VEL
LIN {X 0,Y 656.668,Z 618.867,A -85,B 0,C 180,E1 31796.595,E2 31796.595} C_VEL
LIN {X 0,Y 656.709,Z 618.869,A -85,B 0,C 180,E1 31793.575,E2 31793.575} C_VEL
LIN {X 0,Y 656.621,Z 618.872,A -85,B 0,C 180,E1 31790.689,E2 31790.689} C_VEL
LIN {X 0,Y 656.707,Z 618.867,A -85,B 0,C 180,E1 31787.822,E2 31787.822} C_VEL
LIN {X 0,Y 656.675,Z 618.865,A -85,B 0,C 180,E1 31784.798,E2 31784.798} C_VEL
LIN {X 0,Y 656.689,Z 618.865,A -85,B 0,C 180,E1 31781.863,E2 31781.863} C_VEL
LIN {X 0,Y 656.709,Z 618.866,A -85,B 0,C 180,E1 31778.759,E2 31778.759} C_VEL
LIN {X 0,Y 656.641,Z 618.869,A -85,B 0,C 180,E1 31775.857,E2 31775.857} C_VEL
LIN {X 0,Y 656.661,Z 618.866,A -85,B 0,C 180,E1 31772.794,E2 31772.794} C_VEL
LIN {X 0,Y 656.649,Z 618.869,A -85,B 0,C 180,E1 31770.001,E2 31770.001} C_VEL
LIN {X 0,Y 656.706,Z 618.857,A -85,B 0,C 180,E1 31766.946,E2 31766.946} C_VEL
LIN {X 0,Y 656.703,Z 618.87,A -85,B 0,C 180,E1 31763.795,E2 31763.795} C_VEL
LIN {X 0,Y 656.708,Z 618.861,A -85,B 0,C 180,E1 31760.714,E2 31760.714} C_VEL
LIN {X 0,Y 656.638,Z 618.866,A -85,B 0,C 180,E1 31757.692,E2 31757.692} C_VEL
LIN {X 0,Y 656.671,Z 618.871,A -85,B 0,C 180,E1 31754.866,E2 31754.866} C_VEL
LIN {X 0,Y 656.652,Z 618.867,A -85,B 0,C 180,E1 31751.812,E2 31751.812} C_VEL
LIN {X 0,Y 656.704,Z 618.866,A -85,B 0,C 180,E1 31748.849,E2 31748.849} C_VEL
LIN {X 0,Y 656.696,Z 618.865,A -85,B 0,C 180,E1 31745.782,E2 31745.782} C_VEL
LIN {X 0,Y 656.667,Z 618.866,A -85,B 0,C 180,E1 31742.821,E2 31742.821} C_VEL
LIN {X 0,Y 656.696,Z 618.871,A -85,B 0,C 180,E1 31739.839,E2 31739.839} C_VEL
LIN {X 0,Y 656.624,Z 618.872,A -85,B 0,C 180,E1 31736.967,E2 31736.967} C_VEL
LIN {X 0,Y 656.7,Z 618.865,A -85,B 0,C 180,E1 31733.945,E2 31733.945} C_VEL
LIN {X 0,Y 656.686,Z 618.869,A -85,B 0,C 180,E1 31730.925,E2 31730.925} C_VEL
LIN {X 0,Y 656.706,Z 618.862,A -85,B 0,C 180,E1 31727.725,E2 31727.725} C_VEL
LIN {X 0,Y 656.671,Z 618.87,A -85,B 0,C 180,E1 31724.679,E2 31724.679} C_VEL
LIN {X 0,Y 656.7,Z 618.868,A -85,B 0,C 180,E1 31721.707,E2 31721.707} C_VEL
LIN {X 0,Y 656.707,Z 619.052,A -85,B 0,C 180,E1 31719.453,E2 31719.453} C_VEL
LIN {X 0,Y 660.527,Z 634.094,A -85,B 0,C 180,E1 31718.2,E2 31718.2} C_VEL
LIN {X 0,Y 660.116,Z 677.3,A -85,B 0,C 180,E1 31715.032,E2 31715.032} C_VEL
LIN {X 0,Y 659.661,Z 716.477,A -85,B 0,C 180,E1 31712.14,E2 31712.14} C_VEL
LIN {X 0,Y 659.14,Z 758.613,A -85,B 0,C 180,E1 31709.038,E2 31709.038} C_VEL
LIN {X 0,Y 658.52,Z 799.518,A -85,B 0,C 180,E1 31706.026,E2 31706.026} C_VEL
LIN {X 0,Y 658.315,Z 820.81,A -85,B 0,C 180,E1 31704.478,E2 31704.478} C_VEL
LIN {X 0,Y 658.709,Z 828.61,A -85,B 0,C 180,E1 31704.379,E2 31704.379} C_VEL
LIN {X 0,Y 658.07,Z 962.723,A -85,B 0,C 180,E1 31702.838,E2 31702.838} C_VEL
LIN {X 0,Y 657.95,Z 978.904,A -85,B 0,C 180,E1 31702.488,E2 31702.488} C_VEL
LIN {X 0,Y 657.771,Z 995.317,A -85,B 0,C 180,E1 31701.957,E2 31701.957} C_VEL
LIN {X 0,Y 657.535,Z 1009.879,A -85,B 0,C 180,E1 31701.309,E2 31701.309} C_VEL
LIN {X 0,Y 657.307,Z 1023.658,A -85,B 0,C 180,E1 31700.524,E2 31700.524} C_VEL
LIN {X 0,Y 657.042,Z 1036.254,A -85,B 0,C 180,E1 31699.617,E2 31699.617} C_VEL
LIN {X 0,Y 656.795,Z 1048.132,A -85,B 0,C 180,E1 31698.55,E2 31698.55} C_VEL
LIN {X 0,Y 656.586,Z 1057.868,A -85,B 0,C 180,E1 31697.455,E2 31697.455} C_VEL
LIN {X 0,Y 656.415,Z 1066.834,A -85,B 0,C 180,E1 31696.184,E2 31696.184} C_VEL
LIN {X 0,Y 656.3,Z 1073.684,A -85,B 0,C 180,E1 31694.918,E2 31694.918} C_VEL
LIN {X 0,Y 656.234,Z 1079.356,A -85,B 0,C 180,E1 31693.479,E2 31693.479} C_VEL
LIN {X 0,Y 656.187,Z 1083.132,A -85,B 0,C 180,E1 31691.958,E2 31691.958} C_VEL
LIN {X 0,Y 656.174,Z 1084.835,A -85,B 0,C 180,E1 31690.534,E2 31690.534} C_VEL
LIN {X 0,Y 656.187,Z 1084.697,A -85,B 0,C 180,E1 31689.113,E2 31689.113} C_VEL
LIN {X 0,Y 656.22,Z 1082.866,A -85,B 0,C 180,E1 31687.704,E2 31687.704} C_VEL
LIN {X 0,Y 656.266,Z 1079.179,A -85,B 0,C 180,E1 31686.296,E2 31686.296} C_VEL
LIN {X 0,Y 656.358,Z 1073.611,A -85,B 0,C 180,E1 31684.892,E2 31684.892} C_VEL
LIN {X 0,Y 656.487,Z 1066.36,A -85,B 0,C 180,E1 31683.578,E2 31683.578} C_VEL
LIN {X 0,Y 656.67,Z 1057.635,A -85,B 0,C 180,E1 31682.354,E2 31682.354} C_VEL
LIN {X 0,Y 656.892,Z 1047.296,A -85,B 0,C 180,E1 31681.219,E2 31681.219} C_VEL
LIN {X 0,Y 657.155,Z 1035.41,A -85,B 0,C 180,E1 31680.172,E2 31680.172} C_VEL
LIN {X 0,Y 657.402,Z 1022.247,A -85,B 0,C 180,E1 31679.257,E2 31679.257} C_VEL
LIN {X 0,Y 657.602,Z 1008.89,A -85,B 0,C 180,E1 31678.517,E2 31678.517} C_VEL
LIN {X 0,Y 657.811,Z 994.468,A -85,B 0,C 180,E1 31677.908,E2 31677.908} C_VEL
LIN {X 0,Y 657.954,Z 980.453,A -85,B 0,C 180,E1 31677.464,E2 31677.464} C_VEL
LIN {X 0,Y 658.047,Z 965.246,A -85,B 0,C 180,E1 31677.119,E2 31677.119} C_VEL
LIN {X 0,Y 658.152,Z 928.656,A -85,B 0,C 180,E1 31676.68,E2 31676.68} C_VEL
LIN {X 0,Y 658.582,Z 822.649,A -85,B 0,C 180,E1 31675.448,E2 31675.448} C_VEL
LIN {X 0,Y 659.101,Z 779.203,A -85,B 0,C 180,E1 31672.282,E2 31672.282} C_VEL
LIN {X 0,Y 659.393,Z 744.275,A -85,B 0,C 180,E1 31669.767,E2 31669.767} C_VEL
LIN {X 0,Y 659.681,Z 705.098,A -85,B 0,C 180,E1 31666.991,E2 31666.991} C_VEL
LIN {X 0,Y 659.572,Z 664.262,A -85,B 0,C 180,E1 31664.163,E2 31664.163} C_VEL
LIN {X 0,Y 659.49,Z 629.781,A -85,B 0,C 180,E1 31661.845,E2 31661.845} C_VEL
LIN {X 0,Y 656.683,Z 618.874,A -85,B 0,C 180,E1 31661,E2 31661} C_VEL
LIN {X 0,Y 656.711,Z 618.867,A -85,B 0,C 180,E1 31657.772,E2 31657.772} C_VEL
LIN {X 0,Y 656.681,Z 618.875,A -85,B 0,C 180,E1 31654.667,E2 31654.667} C_VEL
LIN {X 0,Y 656.713,Z 618.869,A -85,B 0,C 180,E1 31651.637,E2 31651.637} C_VEL
LIN {X 0,Y 656.691,Z 618.87,A -85,B 0,C 180,E1 31648.617,E2 31648.617} C_VEL
LIN {X 0,Y 656.705,Z 618.866,A -85,B 0,C 180,E1 31645.393,E2 31645.393} C_VEL
LIN {X 0,Y 656.672,Z 618.871,A -85,B 0,C 180,E1 31642.349,E2 31642.349} C_VEL
LIN {X 0,Y 656.712,Z 618.868,A -85,B 0,C 180,E1 31639.306,E2 31639.306} C_VEL
LIN {X 0,Y 656.697,Z 618.87,A -85,B 0,C 180,E1 31636.193,E2 31636.193} C_VEL
LIN {X 0,Y 656.699,Z 618.866,A -85,B 0,C 180,E1 31633.007,E2 31633.007} C_VEL
LIN {X 0,Y 656.667,Z 618.871,A -85,B 0,C 180,E1 31629.981,E2 31629.981} C_VEL
LIN {X 0,Y 656.712,Z 618.867,A -85,B 0,C 180,E1 31626.86,E2 31626.86} C_VEL
LIN {X 0,Y 656.732,Z 619.033,A -85,B 0,C 180,E1 31625.002,E2 31625.002} C_VEL
LIN {X 0,Y 664.075,Z 642.665,A -85,B 0,C 180,E1 31622.565,E2 31622.565} C_VEL
LIN {X 0,Y 662.886,Z 676.546,A -85,B 0,C 180,E1 31619.801,E2 31619.801} C_VEL
LIN {X 0,Y 662.807,Z 682.391,A -85,B 0,C 180,E1 31619.357,E2 31619.357} C_VEL
LIN {X 0,Y 666.823,Z 702.527,A -85,B 0,C 180,E1 31618.901,E2 31618.901} C_VEL
LIN {X 0,Y 665.597,Z 834.158,A -85,B 0,C 180,E1 31617.359,E2 31617.359} C_VEL
LIN {X 0,Y 664.427,Z 983.504,A -85,B 0,C 180,E1 31615.631,E2 31615.631} C_VEL
LIN {X 0,Y 663.957,Z 1006.161,A -85,B 0,C 180,E1 31615.228,E2 31615.228} C_VEL
LIN {X 0,Y 663.418,Z 1027.478,A -85,B 0,C 180,E1 31614.698,E2 31614.698} C_VEL
LIN {X 0,Y 662.752,Z 1047.929,A -85,B 0,C 180,E1 31614.037,E2 31614.037} C_VEL
LIN {X 0,Y 661.992,Z 1068.358,A -85,B 0,C 180,E1 31613.216,E2 31613.216} C_VEL
LIN {X 0,Y 661.24,Z 1087.257,A -85,B 0,C 180,E1 31612.304,E2 31612.304} C_VEL
LIN {X 0,Y 660.326,Z 1106.595,A -85,B 0,C 180,E1 31611.169,E2 31611.169} C_VEL
LIN {X 0,Y 659.444,Z 1124.449,A -85,B 0,C 180,E1 31609.933,E2 31609.933} C_VEL
LIN {X 0,Y 658.639,Z 1141.651,A -85,B 0,C 180,E1 31608.543,E2 31608.543} C_VEL
LIN {X 0,Y 657.925,Z 1157.486,A -85,B 0,C 180,E1 31607.055,E2 31607.055} C_VEL
LIN {X 0,Y 657.327,Z 1171.328,A -85,B 0,C 180,E1 31605.527,E2 31605.527} C_VEL
LIN {X 0,Y 656.817,Z 1184.552,A -85,B 0,C 180,E1 31603.826,E2 31603.826} C_VEL
LIN {X 0,Y 656.462,Z 1195.751,A -85,B 0,C 180,E1 31602.132,E2 31602.132} C_VEL
LIN {X 0,Y 656.214,Z 1205.516,A -85,B 0,C 180,E1 31600.357,E2 31600.357} C_VEL
LIN {X 0,Y 656.061,Z 1213.824,A -85,B 0,C 180,E1 31598.5,E2 31598.5} C_VEL
LIN {X 0,Y 655.956,Z 1220.388,A -85,B 0,C 180,E1 31596.651,E2 31596.651} C_VEL
LIN {X 0,Y 655.913,Z 1225.228,A -85,B 0,C 180,E1 31594.808,E2 31594.808} C_VEL
LIN {X 0,Y 655.906,Z 1228.562,A -85,B 0,C 180,E1 31592.882,E2 31592.882} C_VEL
LIN {X 0,Y 655.906,Z 1230.237,A -85,B 0,C 180,E1 31591.047,E2 31591.047} C_VEL
LIN {X 0,Y 655.909,Z 1230.304,A -85,B 0,C 180,E1 31589.213,E2 31589.213} C_VEL
LIN {X 0,Y 655.912,Z 1228.784,A -85,B 0,C 180,E1 31587.29,E2 31587.29} C_VEL
LIN {X 0,Y 655.92,Z 1225.628,A -85,B 0,C 180,E1 31585.365,E2 31585.365} C_VEL
LIN {X 0,Y 655.957,Z 1220.888,A -85,B 0,C 180,E1 31583.522,E2 31583.522} C_VEL
LIN {X 0,Y 656.057,Z 1214.167,A -85,B 0,C 180,E1 31581.586,E2 31581.586} C_VEL
LIN {X 0,Y 656.197,Z 1206.417,A -85,B 0,C 180,E1 31579.818,E2 31579.818} C_VEL
LIN {X 0,Y 656.43,Z 1196.77,A -85,B 0,C 180,E1 31578.043,E2 31578.043} C_VEL
LIN {X 0,Y 656.796,Z 1185.17,A -85,B 0,C 180,E1 31576.261,E2 31576.261} C_VEL
LIN {X 0,Y 657.275,Z 1172.847,A -85,B 0,C 180,E1 31574.65,E2 31574.65} C_VEL
LIN {X 0,Y 657.84,Z 1159.16,A -85,B 0,C 180,E1 31573.122,E2 31573.122} C_VEL
LIN {X 0,Y 658.543,Z 1143.457,A -85,B 0,C 180,E1 31571.617,E2 31571.617} C_VEL
LIN {X 0,Y 659.361,Z 1126.35,A -85,B 0,C 180,E1 31570.209,E2 31570.209} C_VEL
LIN {X 0,Y 660.235,Z 1108.727,A -85,B 0,C 180,E1 31568.965,E2 31568.965} C_VEL
LIN {X 0,Y 661.109,Z 1089.655,A -85,B 0,C 180,E1 31567.829,E2 31567.829} C_VEL
LIN {X 0,Y 661.886,Z 1070.91,A -85,B 0,C 180,E1 31566.902,E2 31566.902} C_VEL
LIN {X 0,Y 662.58,Z 1051.149,A -85,B 0,C 180,E1 31566.096,E2 31566.096} C_VEL
LIN {X 0,Y 663.218,Z 1030.106,A -85,B 0,C 180,E1 31565.41,E2 31565.41} C_VEL
LIN {X 0,Y 663.764,Z 1007.147,A -85,B 0,C 180,E1 31564.831,E2 31564.831} C_VEL
LIN {X 0,Y 664.213,Z 985.039,A -85,B 0,C 180,E1 31564.433,E2 31564.433} C_VEL
LIN {X 0,Y 665.716,Z 790.042,A -85,B 0,C 180,E1 31562.179,E2 31562.179} C_VEL
LIN {X 0,Y 666.484,Z 700.496,A -85,B 0,C 180,E1 31561.09,E2 31561.09} C_VEL
LIN {X 0,Y 662.284,Z 679.482,A -85,B 0,C 180,E1 31560.592,E2 31560.592} C_VEL
LIN {X 0,Y 663.356,Z 643.911,A -85,B 0,C 180,E1 31557.739,E2 31557.739} C_VEL
LIN {X 0,Y 663.139,Z 640.558,A -85,B 0,C 180,E1 31557.446,E2 31557.446} C_VEL
LIN {X 0,Y 657.876,Z 622.9,A -85,B 0,C 180,E1 31555.62,E2 31555.62} C_VEL
LIN {X 0,Y 656.701,Z 618.869,A -85,B 0,C 180,E1 31555.154,E2 31555.154} C_VEL
LIN {X 0,Y 656.689,Z 618.871,A -85,B 0,C 180,E1 31551.926,E2 31551.926} C_VEL
LIN {X 0,Y 656.708,Z 618.865,A -85,B 0,C 180,E1 31548.87,E2 31548.87} C_VEL
LIN {X 0,Y 656.676,Z 618.872,A -85,B 0,C 180,E1 31545.698,E2 31545.698} C_VEL
LIN {X 0,Y 656.705,Z 618.866,A -85,B 0,C 180,E1 31542.654,E2 31542.654} C_VEL
LIN {X 0,Y 656.665,Z 618.873,A -85,B 0,C 180,E1 31539.603,E2 31539.603} C_VEL
LIN {X 0,Y 656.682,Z 618.868,A -85,B 0,C 180,E1 31536.757,E2 31536.757} C_VEL
LIN {X 0,Y 656.662,Z 618.874,A -85,B 0,C 180,E1 31533.556,E2 31533.556} C_VEL
LIN {X 0,Y 656.66,Z 618.873,A -85,B 0,C 180,E1 31530.774,E2 31530.774} C_VEL
LIN {X 0,Y 656.68,Z 618.94,A -85,B 0,C 180,E1 31530.65,E2 31530.65} C_VEL
LIN {X 0,Y 659.566,Z 628.436,A -85,B 0,C 180,E1 31529.454,E2 31529.454} C_VEL
LIN {X 0,Y 666.634,Z 642.757,A -85,B 0,C 180,E1 31528.898,E2 31528.898} C_VEL
LIN {X 0,Y 666.938,Z 646.5,A -85,B 0,C 180,E1 31528.834,E2 31528.834} C_VEL
LIN {X 0,Y 665.156,Z 811.612,A -85,B 0,C 180,E1 31526.845,E2 31526.845} C_VEL
LIN {X 0,Y 664.28,Z 928.278,A -85,B 0,C 180,E1 31525.497,E2 31525.497} C_VEL
LIN {X 0,Y 663.814,Z 950.661,A -85,B 0,C 180,E1 31525.075,E2 31525.075} C_VEL
LIN {X 0,Y 663.255,Z 972.223,A -85,B 0,C 180,E1 31524.509,E2 31524.509} C_VEL
LIN {X 0,Y 662.581,Z 992.912,A -85,B 0,C 180,E1 31523.81,E2 31523.81} C_VEL
LIN {X 0,Y 661.857,Z 1012.571,A -85,B 0,C 180,E1 31522.989,E2 31522.989} C_VEL
LIN {X 0,Y 661.067,Z 1030.482,A -85,B 0,C 180,E1 31522.079,E2 31522.079} C_VEL
LIN {X 0,Y 660.153,Z 1050.033,A -85,B 0,C 180,E1 31520.899,E2 31520.899} C_VEL
LIN {X 0,Y 659.313,Z 1067.715,A -85,B 0,C 180,E1 31519.646,E2 31519.646} C_VEL
LIN {X 0,Y 658.49,Z 1084.727,A -85,B 0,C 180,E1 31518.23,E2 31518.23} C_VEL
LIN {X 0,Y 657.799,Z 1100.054,A -85,B 0,C 180,E1 31516.737,E2 31516.737} C_VEL
LIN {X 0,Y 657.193,Z 1114.644,A -85,B 0,C 180,E1 31515.082,E2 31515.082} C_VEL
LIN {X 0,Y 656.738,Z 1127.421,A -85,B 0,C 180,E1 31513.382,E2 31513.382} C_VEL
LIN {X 0,Y 656.391,Z 1138.586,A -85,B 0,C 180,E1 31511.602,E2 31511.602} C_VEL
LIN {X 0,Y 656.16,Z 1148.255,A -85,B 0,C 180,E1 31509.74,E2 31509.74} C_VEL
LIN {X 0,Y 656.019,Z 1156.064,A -85,B 0,C 180,E1 31507.886,E2 31507.886} C_VEL
LIN {X 0,Y 655.942,Z 1162.042,A -85,B 0,C 180,E1 31506.039,E2 31506.039} C_VEL
LIN {X 0,Y 655.908,Z 1166.533,A -85,B 0,C 180,E1 31504.11,E2 31504.11} C_VEL
LIN {X 0,Y 655.901,Z 1169.287,A -85,B 0,C 180,E1 31502.273,E2 31502.273} C_VEL
LIN {X 0,Y 655.899,Z 1170.382,A -85,B 0,C 180,E1 31500.439,E2 31500.439} C_VEL
LIN {X 0,Y 655.905,Z 1169.923,A -85,B 0,C 180,E1 31498.43,E2 31498.43} C_VEL
LIN {X 0,Y 655.917,Z 1167.814,A -85,B 0,C 180,E1 31496.506,E2 31496.506} C_VEL
LIN {X 0,Y 655.938,Z 1164.098,A -85,B 0,C 180,E1 31494.667,E2 31494.667} C_VEL
LIN {X 0,Y 655.99,Z 1158.552,A -85,B 0,C 180,E1 31492.734,E2 31492.734} C_VEL
LIN {X 0,Y 656.1,Z 1151.502,A -85,B 0,C 180,E1 31490.883,E2 31490.883} C_VEL
LIN {X 0,Y 656.272,Z 1142.994,A -85,B 0,C 180,E1 31489.112,E2 31489.112} C_VEL
LIN {X 0,Y 656.56,Z 1132.717,A -85,B 0,C 180,E1 31487.334,E2 31487.334} C_VEL
LIN {X 0,Y 656.959,Z 1120.995,A -85,B 0,C 180,E1 31485.638,E2 31485.638} C_VEL
LIN {X 0,Y 657.466,Z 1107.845,A -85,B 0,C 180,E1 31484.024,E2 31484.024} C_VEL
LIN {X 0,Y 658.092,Z 1093.402,A -85,B 0,C 180,E1 31482.495,E2 31482.495} C_VEL
LIN {X 0,Y 658.876,Z 1076.764,A -85,B 0,C 180,E1 31480.988,E2 31480.988} C_VEL
LIN {X 0,Y 659.711,Z 1059.333,A -85,B 0,C 180,E1 31479.647,E2 31479.647} C_VEL
LIN {X 0,Y 660.553,Z 1041.464,A -85,B 0,C 180,E1 31478.469,E2 31478.469} C_VEL
LIN {X 0,Y 661.433,Z 1022.871,A -85,B 0,C 180,E1 31477.423,E2 31477.423} C_VEL
LIN {X 0,Y 662.222,Z 1003.394,A -85,B 0,C 180,E1 31476.511,E2 31476.511} C_VEL
LIN {X 0,Y 662.974,Z 983.126,A -85,B 0,C 180,E1 31475.736,E2 31475.736} C_VEL
LIN {X 0,Y 663.663,Z 960.977,A -85,B 0,C 180,E1 31475.064,E2 31475.064} C_VEL
LIN {X 0,Y 664.205,Z 939.204,A -85,B 0,C 180,E1 31474.568,E2 31474.568} C_VEL
LIN {X 0,Y 664.568,Z 916.793,A -85,B 0,C 180,E1 31474.224,E2 31474.224} C_VEL
LIN {X 0,Y 664.985,Z 866.827,A -85,B 0,C 180,E1 31473.647,E2 31473.647} C_VEL
LIN {X 0,Y 664.137,Z 859.237,A -85,B 0,C 180,E1 31473.526,E2 31473.526} C_VEL
LIN {X 0,Y 658.605,Z 839.402,A -85,B 0,C 180,E1 31473.07,E2 31473.07} C_VEL
LIN {X 0,Y 657.985,Z 832.877,A -85,B 0,C 180,E1 31472.968,E2 31472.968} C_VEL
LIN {X 0,Y 659.89,Z 645.589,A -85,B 0,C 180,E1 31470.717,E2 31470.717} C_VEL
LIN {X 0,Y 650.295,Z 625.516,A -85,B 0,C 180,E1 31469.96,E2 31469.96} C_VEL
LIN {X 0,Y 648.701,Z 619.866,A -85,B 0,C 180,E1 31469.28,E2 31469.28} C_VEL
LIN {X 0,Y 648.714,Z 619.863,A -85,B 0,C 180,E1 31466.18,E2 31466.18} C_VEL
LIN {X 0,Y 648.721,Z 619.859,A -85,B 0,C 180,E1 31463.384,E2 31463.384} C_VEL
LIN {X 0,Y 648.76,Z 619.85,A -85,B 0,C 180,E1 31460.241,E2 31460.241} C_VEL
LIN {X 0,Y 648.756,Z 619.857,A -85,B 0,C 180,E1 31457.185,E2 31457.185} C_VEL
LIN {X 0,Y 648.774,Z 619.854,A -85,B 0,C 180,E1 31454.034,E2 31454.034} C_VEL
LIN {X 0,Y 648.693,Z 619.86,A -85,B 0,C 180,E1 31451.089,E2 31451.089} C_VEL
LIN {X 0,Y 648.763,Z 619.858,A -85,B 0,C 180,E1 31448.173,E2 31448.173} C_VEL
LIN {X 0,Y 648.715,Z 619.856,A -85,B 0,C 180,E1 31445.203,E2 31445.203} C_VEL
LIN {X 0,Y 648.765,Z 619.853,A -85,B 0,C 180,E1 31442.212,E2 31442.212} C_VEL
LIN {X 0,Y 648.767,Z 619.856,A -85,B 0,C 180,E1 31439.095,E2 31439.095} C_VEL
LIN {X 0,Y 648.739,Z 619.852,A -85,B 0,C 180,E1 31436.037,E2 31436.037} C_VEL
LIN {X 0,Y 648.697,Z 619.859,A -85,B 0,C 180,E1 31432.858,E2 31432.858} C_VEL
LIN {X 0,Y 648.711,Z 619.861,A -85,B 0,C 180,E1 31430.105,E2 31430.105} C_VEL
LIN {X 0,Y 648.728,Z 619.854,A -85,B 0,C 180,E1 31427.03,E2 31427.03} C_VEL
LIN {X 0,Y 648.771,Z 619.853,A -85,B 0,C 180,E1 31424.095,E2 31424.095} C_VEL
LIN {X 0,Y 648.761,Z 619.854,A -85,B 0,C 180,E1 31420.929,E2 31420.929} C_VEL
LIN {X 0,Y 648.721,Z 619.853,A -85,B 0,C 180,E1 31417.975,E2 31417.975} C_VEL
LIN {X 0,Y 648.761,Z 619.86,A -85,B 0,C 180,E1 31414.952,E2 31414.952} C_VEL
LIN {X 0,Y 648.69,Z 619.855,A -85,B 0,C 180,E1 31411.944,E2 31411.944} C_VEL
LIN {X 0,Y 648.765,Z 619.852,A -85,B 0,C 180,E1 31408.942,E2 31408.942} C_VEL
LIN {X 0,Y 648.759,Z 619.852,A -85,B 0,C 180,E1 31405.847,E2 31405.847} C_VEL
LIN {X 0,Y 648.769,Z 619.85,A -85,B 0,C 180,E1 31402.652,E2 31402.652} C_VEL
LIN {X 0,Y 648.718,Z 619.851,A -85,B 0,C 180,E1 31399.612,E2 31399.612} C_VEL
LIN {X 0,Y 648.763,Z 619.854,A -85,B 0,C 180,E1 31396.635,E2 31396.635} C_VEL
LIN {X 0,Y 648.692,Z 619.858,A -85,B 0,C 180,E1 31393.617,E2 31393.617} C_VEL
LIN {X 0,Y 648.772,Z 619.853,A -85,B 0,C 180,E1 31390.65,E2 31390.65} C_VEL
LIN {X 0,Y 648.754,Z 619.857,A -85,B 0,C 180,E1 31387.53,E2 31387.53} C_VEL
LIN {X 0,Y 648.765,Z 619.85,A -85,B 0,C 180,E1 31384.364,E2 31384.364} C_VEL
LIN {X 0,Y 648.72,Z 619.859,A -85,B 0,C 180,E1 31381.258,E2 31381.258} C_VEL
LIN {X 0,Y 648.72,Z 619.859,A -85,B 0,C 180,E1 31378.463,E2 31378.463} C_VEL
LIN {X 0,Y 648.698,Z 619.859,A -85,B 0,C 180,E1 31375.338,E2 31375.338} C_VEL
LIN {X 0,Y 648.765,Z 619.86,A -85,B 0,C 180,E1 31372.501,E2 31372.501} C_VEL
LIN {X 0,Y 648.75,Z 619.854,A -85,B 0,C 180,E1 31369.43,E2 31369.43} C_VEL
LIN {X 0,Y 648.74,Z 619.856,A -85,B 0,C 180,E1 31366.415,E2 31366.415} C_VEL
LIN {X 0,Y 648.766,Z 619.857,A -85,B 0,C 180,E1 31363.298,E2 31363.298} C_VEL
LIN {X 0,Y 648.684,Z 619.865,A -85,B 0,C 180,E1 31360.458,E2 31360.458} C_VEL
LIN {X 0,Y 648.755,Z 619.917,A -85,B 0,C 180,E1 31359.701,E2 31359.701} C_VEL
LIN {X 0,Y 652.922,Z 636.207,A -85,B 0,C 180,E1 31358.329,E2 31358.329} C_VEL
LIN {X 0,Y 652.445,Z 681.077,A -85,B 0,C 180,E1 31355.022,E2 31355.022} C_VEL
LIN {X 0,Y 651.965,Z 721.289,A -85,B 0,C 180,E1 31352.046,E2 31352.046} C_VEL
LIN {X 0,Y 651.333,Z 764.869,A -85,B 0,C 180,E1 31348.816,E2 31348.816} C_VEL
LIN {X 0,Y 650.723,Z 805.725,A -85,B 0,C 180,E1 31345.789,E2 31345.789} C_VEL
LIN {X 0,Y 650.574,Z 821.643,A -85,B 0,C 180,E1 31344.644,E2 31344.644} C_VEL
LIN {X 0,Y 650.954,Z 829.304,A -85,B 0,C 180,E1 31344.545,E2 31344.545} C_VEL
LIN {X 0,Y 650.251,Z 963.639,A -85,B 0,C 180,E1 31342.975,E2 31342.975} C_VEL
LIN {X 0,Y 650.129,Z 979.825,A -85,B 0,C 180,E1 31342.619,E2 31342.619} C_VEL
LIN {X 0,Y 649.951,Z 995.596,A -85,B 0,C 180,E1 31342.105,E2 31342.105} C_VEL
LIN {X 0,Y 649.716,Z 1009.673,A -85,B 0,C 180,E1 31341.483,E2 31341.483} C_VEL
LIN {X 0,Y 649.457,Z 1024.407,A -85,B 0,C 180,E1 31340.642,E2 31340.642} C_VEL
LIN {X 0,Y 649.171,Z 1037.207,A -85,B 0,C 180,E1 31339.711,E2 31339.711} C_VEL
LIN {X 0,Y 648.906,Z 1049.12,A -85,B 0,C 180,E1 31338.629,E2 31338.629} C_VEL
LIN {X 0,Y 648.676,Z 1059.085,A -85,B 0,C 180,E1 31337.49,E2 31337.49} C_VEL
LIN {X 0,Y 648.493,Z 1068.012,A -85,B 0,C 180,E1 31336.203,E2 31336.203} C_VEL
LIN {X 0,Y 648.366,Z 1074.794,A -85,B 0,C 180,E1 31334.922,E2 31334.922} C_VEL
LIN {X 0,Y 648.296,Z 1080.127,A -85,B 0,C 180,E1 31333.556,E2 31333.556} C_VEL
LIN {X 0,Y 648.242,Z 1084.151,A -85,B 0,C 180,E1 31331.926,E2 31331.926} C_VEL
LIN {X 0,Y 648.228,Z 1085.789,A -85,B 0,C 180,E1 31330.485,E2 31330.485} C_VEL
LIN {X 0,Y 648.248,Z 1085.542,A -85,B 0,C 180,E1 31328.96,E2 31328.96} C_VEL
LIN {X 0,Y 648.282,Z 1083.512,A -85,B 0,C 180,E1 31327.531,E2 31327.531} C_VEL
LIN {X 0,Y 648.349,Z 1079.355,A -85,B 0,C 180,E1 31326.018,E2 31326.018} C_VEL
LIN {X 0,Y 648.453,Z 1073.829,A -85,B 0,C 180,E1 31324.686,E2 31324.686} C_VEL
LIN {X 0,Y 648.607,Z 1066.377,A -85,B 0,C 180,E1 31323.356,E2 31323.356} C_VEL
LIN {X 0,Y 648.792,Z 1058.068,A -85,B 0,C 180,E1 31322.206,E2 31322.206} C_VEL
LIN {X 0,Y 649.043,Z 1047.603,A -85,B 0,C 180,E1 31321.057,E2 31321.057} C_VEL
LIN {X 0,Y 649.313,Z 1036.07,A -85,B 0,C 180,E1 31320.042,E2 31320.042} C_VEL
LIN {X 0,Y 649.578,Z 1022.82,A -85,B 0,C 180,E1 31319.116,E2 31319.116} C_VEL
LIN {X 0,Y 649.791,Z 1009.315,A -85,B 0,C 180,E1 31318.367,E2 31318.367} C_VEL
LIN {X 0,Y 649.995,Z 995.913,A -85,B 0,C 180,E1 31317.794,E2 31317.794} C_VEL
LIN {X 0,Y 650.145,Z 981.524,A -85,B 0,C 180,E1 31317.332,E2 31317.332} C_VEL
LIN {X 0,Y 650.235,Z 966.394,A -85,B 0,C 180,E1 31316.983,E2 31316.983} C_VEL
LIN {X 0,Y 650.349,Z 929.861,A -85,B 0,C 180,E1 31316.537,E2 31316.537} C_VEL
LIN {X 0,Y 650.885,Z 823.789,A -85,B 0,C 180,E1 31315.284,E2 31315.284} C_VEL
LIN {X 0,Y 651.426,Z 782.132,A -85,B 0,C 180,E1 31312.235,E2 31312.235} C_VEL
LIN {X 0,Y 651.778,Z 742.72,A -85,B 0,C 180,E1 31309.39,E2 31309.39} C_VEL
LIN {X 0,Y 652.048,Z 704.764,A -85,B 0,C 180,E1 31306.7,E2 31306.7} C_VEL
LIN {X 0,Y 651.971,Z 665.548,A -85,B 0,C 180,E1 31303.973,E2 31303.973} C_VEL
LIN {X 0,Y 651.831,Z 631.548,A -85,B 0,C 180,E1 31301.67,E2 31301.67} C_VEL
LIN {X 0,Y 648.732,Z 619.863,A -85,B 0,C 180,E1 31300.786,E2 31300.786} C_VEL
LIN {X 0,Y 648.764,Z 619.859,A -85,B 0,C 180,E1 31297.527,E2 31297.527} C_VEL
LIN {X 0,Y 648.767,Z 619.862,A -85,B 0,C 180,E1 31294.366,E2 31294.366} C_VEL
LIN {X 0,Y 648.739,Z 619.86,A -85,B 0,C 180,E1 31291.256,E2 31291.256} C_VEL
LIN {X 0,Y 648.74,Z 619.859,A -85,B 0,C 180,E1 31288.395,E2 31288.395} C_VEL
LIN {X 0,Y 648.76,Z 619.857,A -85,B 0,C 180,E1 31285.075,E2 31285.075} C_VEL
LIN {X 0,Y 648.764,Z 619.858,A -85,B 0,C 180,E1 31281.938,E2 31281.938} C_VEL
LIN {X 0,Y 648.745,Z 619.859,A -85,B 0,C 180,E1 31278.907,E2 31278.907} C_VEL
LIN {X 0,Y 648.747,Z 619.858,A -85,B 0,C 180,E1 31275.906,E2 31275.906} C_VEL
LIN {X 0,Y 648.753,Z 619.856,A -85,B 0,C 180,E1 31272.676,E2 31272.676} C_VEL
LIN {X 0,Y 648.743,Z 619.86,A -85,B 0,C 180,E1 31269.726,E2 31269.726} C_VEL
LIN {X 0,Y 648.769,Z 619.859,A -85,B 0,C 180,E1 31266.724,E2 31266.724} C_VEL
LIN {X 0,Y 648.774,Z 619.979,A -85,B 0,C 180,E1 31265.382,E2 31265.382} C_VEL
LIN {X 0,Y 656.347,Z 644.191,A -85,B 0,C 180,E1 31262.841,E2 31262.841} C_VEL
LIN {X 0,Y 656.678,Z 647.238,A -85,B 0,C 180,E1 31262.563,E2 31262.563} C_VEL
LIN {X 0,Y 655.366,Z 681.89,A -85,B 0,C 180,E1 31259.726,E2 31259.726} C_VEL
LIN {X 0,Y 659.779,Z 703.91,A -85,B 0,C 180,E1 31259.216,E2 31259.216} C_VEL
LIN {X 0,Y 658.447,Z 829.418,A -85,B 0,C 180,E1 31257.72,E2 31257.72} C_VEL
LIN {X 0,Y 657.06,Z 982.519,A -85,B 0,C 180,E1 31255.916,E2 31255.916} C_VEL
LIN {X 0,Y 656.559,Z 1005.383,A -85,B 0,C 180,E1 31255.508,E2 31255.508} C_VEL
LIN {X 0,Y 655.962,Z 1026.769,A -85,B 0,C 180,E1 31254.974,E2 31254.974} C_VEL
LIN {X 0,Y 655.221,Z 1047.907,A -85,B 0,C 180,E1 31254.283,E2 31254.283} C_VEL
LIN {X 0,Y 654.395,Z 1068.252,A -85,B 0,C 180,E1 31253.454,E2 31253.454} C_VEL
LIN {X 0,Y 653.53,Z 1088.403,A -85,B 0,C 180,E1 31252.464,E2 31252.464} C_VEL
LIN {X 0,Y 652.631,Z 1107.851,A -85,B 0,C 180,E1 31251.326,E2 31251.326} C_VEL
LIN {X 0,Y 651.806,Z 1124.27,A -85,B 0,C 180,E1 31250.19,E2 31250.19} C_VEL
LIN {X 0,Y 650.94,Z 1141.143,A -85,B 0,C 180,E1 31248.817,E2 31248.817} C_VEL
LIN {X 0,Y 650.168,Z 1156.58,A -85,B 0,C 180,E1 31247.357,E2 31247.357} C_VEL
LIN {X 0,Y 649.502,Z 1170.583,A -85,B 0,C 180,E1 31245.808,E2 31245.808} C_VEL
LIN {X 0,Y 648.945,Z 1183.916,A -85,B 0,C 180,E1 31244.088,E2 31244.088} C_VEL
LIN {X 0,Y 648.55,Z 1195.234,A -85,B 0,C 180,E1 31242.373,E2 31242.373} C_VEL
LIN {X 0,Y 648.264,Z 1205.056,A -85,B 0,C 180,E1 31240.575,E2 31240.575} C_VEL
LIN {X 0,Y 648.075,Z 1213.471,A -85,B 0,C 180,E1 31238.695,E2 31238.695} C_VEL
LIN {X 0,Y 647.964,Z 1220.133,A -85,B 0,C 180,E1 31236.823,E2 31236.823} C_VEL
LIN {X 0,Y 647.915,Z 1225.023,A -85,B 0,C 180,E1 31234.956,E2 31234.956} C_VEL
LIN {X 0,Y 647.903,Z 1228.448,A -85,B 0,C 180,E1 31233.006,E2 31233.006} C_VEL
LIN {X 0,Y 647.903,Z 1230.21,A -85,B 0,C 180,E1 31231.148,E2 31231.148} C_VEL
LIN {X 0,Y 647.906,Z 1230.326,A -85,B 0,C 180,E1 31229.291,E2 31229.291} C_VEL
LIN {X 0,Y 647.911,Z 1228.783,A -85,B 0,C 180,E1 31227.257,E2 31227.257} C_VEL
LIN {X 0,Y 647.918,Z 1225.628,A -85,B 0,C 180,E1 31225.307,E2 31225.307} C_VEL
LIN {X 0,Y 647.959,Z 1220.888,A -85,B 0,C 180,E1 31223.442,E2 31223.442} C_VEL
LIN {X 0,Y 648.069,Z 1214.167,A -85,B 0,C 180,E1 31221.481,E2 31221.481} C_VEL
LIN {X 0,Y 648.228,Z 1206.417,A -85,B 0,C 180,E1 31219.692,E2 31219.692} C_VEL
LIN {X 0,Y 648.499,Z 1196.432,A -85,B 0,C 180,E1 31217.836,E2 31217.836} C_VEL
LIN {X 0,Y 648.893,Z 1185.169,A -85,B 0,C 180,E1 31216.09,E2 31216.09} C_VEL
LIN {X 0,Y 649.417,Z 1172.846,A -85,B 0,C 180,E1 31214.459,E2 31214.459} C_VEL
LIN {X 0,Y 650.042,Z 1159.158,A -85,B 0,C 180,E1 31212.914,E2 31212.914} C_VEL
LIN {X 0,Y 650.784,Z 1144.009,A -85,B 0,C 180,E1 31211.441,E2 31211.441} C_VEL
LIN {X 0,Y 651.656,Z 1127.28,A -85,B 0,C 180,E1 31210.037,E2 31210.037} C_VEL
LIN {X 0,Y 652.345,Z 1113.129,A -85,B 0,C 180,E1 31209.028,E2 31209.028} C_VEL
LIN {X 0,Y 653.196,Z 1094.208,A -85,B 0,C 180,E1 31207.878,E2 31207.878} C_VEL
LIN {X 0,Y 654.049,Z 1074.472,A -85,B 0,C 180,E1 31206.864,E2 31206.864} C_VEL
LIN {X 0,Y 654.814,Z 1053.647,A -85,B 0,C 180,E1 31205.986,E2 31205.986} C_VEL
LIN {X 0,Y 655.541,Z 1031.956,A -85,B 0,C 180,E1 31205.247,E2 31205.247} C_VEL
LIN {X 0,Y 656.129,Z 1010.24,A -85,B 0,C 180,E1 31204.669,E2 31204.669} C_VEL
LIN {X 0,Y 656.635,Z 988.047,A -85,B 0,C 180,E1 31204.242,E2 31204.242} C_VEL
LIN {X 0,Y 657.063,Z 944.929,A -85,B 0,C 180,E1 31203.716,E2 31203.716} C_VEL
LIN {X 0,Y 658.421,Z 788.04,A -85,B 0,C 180,E1 31201.873,E2 31201.873} C_VEL
LIN {X 0,Y 659.443,Z 701.983,A -85,B 0,C 180,E1 31200.779,E2 31200.779} C_VEL
LIN {X 0,Y 654.798,Z 678.721,A -85,B 0,C 180,E1 31200.22,E2 31200.22} C_VEL
LIN {X 0,Y 656.035,Z 644.302,A -85,B 0,C 180,E1 31197.398,E2 31197.398} C_VEL
LIN {X 0,Y 650.814,Z 626.464,A -85,B 0,C 180,E1 31195.515,E2 31195.515} C_VEL
LIN {X 0,Y 648.763,Z 619.859,A -85,B 0,C 180,E1 31194.731,E2 31194.731} C_VEL
LIN {X 0,Y 648.739,Z 619.861,A -85,B 0,C 180,E1 31191.677,E2 31191.677} C_VEL
LIN {X 0,Y 648.767,Z 619.857,A -85,B 0,C 180,E1 31188.609,E2 31188.609} C_VEL
LIN {X 0,Y 648.732,Z 619.86,A -85,B 0,C 180,E1 31185.532,E2 31185.532} C_VEL
LIN {X 0,Y 648.768,Z 619.856,A -85,B 0,C 180,E1 31182.548,E2 31182.548} C_VEL
LIN {X 0,Y 648.723,Z 619.862,A -85,B 0,C 180,E1 31179.538,E2 31179.538} C_VEL
LIN {X 0,Y 648.759,Z 619.857,A -85,B 0,C 180,E1 31176.583,E2 31176.583} C_VEL
LIN {X 0,Y 648.719,Z 619.863,A -85,B 0,C 180,E1 31173.492,E2 31173.492} C_VEL
LIN {X 0,Y 648.742,Z 620.109,A -85,B 0,C 180,E1 31171.088,E2 31171.088} C_VEL
LIN {X 0,Y 651.698,Z 629.416,A -85,B 0,C 180,E1 31169.858,E2 31169.858} C_VEL
LIN {X 0,Y 659.784,Z 645.428,A -85,B 0,C 180,E1 31169.2,E2 31169.2} C_VEL
LIN {X 0,Y 658.372,Z 759.855,A -85,B 0,C 180,E1 31167.745,E2 31167.745} C_VEL
LIN {X 0,Y 656.799,Z 929.414,A -85,B 0,C 180,E1 31165.733,E2 31165.733} C_VEL
LIN {X 0,Y 656.317,Z 951.71,A -85,B 0,C 180,E1 31165.303,E2 31165.303} C_VEL
LIN {X 0,Y 655.721,Z 973.3,A -85,B 0,C 180,E1 31164.726,E2 31164.726} C_VEL
LIN {X 0,Y 655.002,Z 994.208,A -85,B 0,C 180,E1 31164.007,E2 31164.007} C_VEL
LIN {X 0,Y 654.198,Z 1014.736,A -85,B 0,C 180,E1 31163.131,E2 31163.131} C_VEL
LIN {X 0,Y 653.313,Z 1034.152,A -85,B 0,C 180,E1 31162.119,E2 31162.119} C_VEL
LIN {X 0,Y 652.403,Z 1052.645,A -85,B 0,C 180,E1 31160.971,E2 31160.971} C_VEL
LIN {X 0,Y 651.518,Z 1070.035,A -85,B 0,C 180,E1 31159.7,E2 31159.7} C_VEL
LIN {X 0,Y 650.679,Z 1086.254,A -85,B 0,C 180,E1 31158.317,E2 31158.317} C_VEL
LIN {X 0,Y 649.937,Z 1101.296,A -85,B 0,C 180,E1 31156.813,E2 31156.813} C_VEL
LIN {X 0,Y 649.296,Z 1115.362,A -85,B 0,C 180,E1 31155.178,E2 31155.178} C_VEL
LIN {X 0,Y 648.805,Z 1127.874,A -85,B 0,C 180,E1 31153.479,E2 31153.479} C_VEL
LIN {X 0,Y 648.44,Z 1138.767,A -85,B 0,C 180,E1 31151.715,E2 31151.715} C_VEL
LIN {X 0,Y 648.186,Z 1148.255,A -85,B 0,C 180,E1 31149.861,E2 31149.861} C_VEL
LIN {X 0,Y 648.033,Z 1156.064,A -85,B 0,C 180,E1 31147.984,E2 31147.984} C_VEL
LIN {X 0,Y 647.949,Z 1162.044,A -85,B 0,C 180,E1 31146.114,E2 31146.114} C_VEL
LIN {X 0,Y 647.911,Z 1166.532,A -85,B 0,C 180,E1 31144.161,E2 31144.161} C_VEL
LIN {X 0,Y 647.901,Z 1169.287,A -85,B 0,C 180,E1 31142.301,E2 31142.301} C_VEL
LIN {X 0,Y 647.899,Z 1170.382,A -85,B 0,C 180,E1 31140.444,E2 31140.444} C_VEL
LIN {X 0,Y 647.903,Z 1169.991,A -85,B 0,C 180,E1 31138.499,E2 31138.499} C_VEL
LIN {X 0,Y 647.917,Z 1168.044,A -85,B 0,C 180,E1 31136.64,E2 31136.64} C_VEL
LIN {X 0,Y 647.939,Z 1164.306,A -85,B 0,C 180,E1 31134.689,E2 31134.689} C_VEL
LIN {X 0,Y 647.995,Z 1158.854,A -85,B 0,C 180,E1 31132.733,E2 31132.733} C_VEL
LIN {X 0,Y 648.109,Z 1151.979,A -85,B 0,C 180,E1 31130.889,E2 31130.889} C_VEL
LIN {X 0,Y 648.301,Z 1143.457,A -85,B 0,C 180,E1 31129.067,E2 31129.067} C_VEL
LIN {X 0,Y 648.612,Z 1133.293,A -85,B 0,C 180,E1 31127.267,E2 31127.267} C_VEL
LIN {X 0,Y 649.041,Z 1121.637,A -85,B 0,C 180,E1 31125.55,E2 31125.55} C_VEL
LIN {X 0,Y 649.593,Z 1108.626,A -85,B 0,C 180,E1 31123.917,E2 31123.917} C_VEL
LIN {X 0,Y 650.273,Z 1094.336,A -85,B 0,C 180,E1 31122.37,E2 31122.37} C_VEL
LIN {X 0,Y 651.1,Z 1077.995,A -85,B 0,C 180,E1 31120.863,E2 31120.863} C_VEL
LIN {X 0,Y 651.978,Z 1061.168,A -85,B 0,C 180,E1 31119.536,E2 31119.536} C_VEL
LIN {X 0,Y 652.906,Z 1042.758,A -85,B 0,C 180,E1 31118.297,E2 31118.297} C_VEL
LIN {X 0,Y 653.829,Z 1024.273,A -85,B 0,C 180,E1 31117.24,E2 31117.24} C_VEL
LIN {X 0,Y 654.713,Z 1003.926,A -85,B 0,C 180,E1 31116.273,E2 31116.273} C_VEL
LIN {X 0,Y 655.536,Z 983.075,A -85,B 0,C 180,E1 31115.467,E2 31115.467} C_VEL
LIN {X 0,Y 656.288,Z 960.468,A -85,B 0,C 180,E1 31114.778,E2 31114.778} C_VEL
LIN {X 0,Y 656.853,Z 938.296,A -85,B 0,C 180,E1 31114.276,E2 31114.276} C_VEL
LIN {X 0,Y 657.257,Z 915.614,A -85,B 0,C 180,E1 31113.93,E2 31113.93} C_VEL
LIN {X 0,Y 657.985,Z 832.877,A -85,B 0,C 180,E1 31112.968,E2 31112.968} C_VEL
LIN {X 0,Y 657.151,Z 825.289,A -85,B 0,C 180,E1 31112.843,E2 31112.843} C_VEL
LIN {X 0,Y 651.69,Z 805.479,A -85,B 0,C 180,E1 31112.366,E2 31112.366} C_VEL
LIN {X 0,Y 651.118,Z 798.959,A -85,B 0,C 180,E1 31112.259,E2 31112.259} C_VEL
LIN {X 0,Y 652.881,Z 647.972,A -85,B 0,C 180,E1 31110.403,E2 31110.403} C_VEL
LIN {X 0,Y 642.175,Z 625.919,A -85,B 0,C 180,E1 31109.551,E2 31109.551} C_VEL
LIN {X 0,Y 640.786,Z 620.854,A -85,B 0,C 180,E1 31108.945,E2 31108.945} C_VEL
LIN {X 0,Y 640.753,Z 620.853,A -85,B 0,C 180,E1 31105.799,E2 31105.799} C_VEL
LIN {X 0,Y 640.83,Z 620.847,A -85,B 0,C 180,E1 31102.858,E2 31102.858} C_VEL
LIN {X 0,Y 640.804,Z 620.843,A -85,B 0,C 180,E1 31099.732,E2 31099.732} C_VEL
LIN {X 0,Y 640.808,Z 620.842,A -85,B 0,C 180,E1 31096.768,E2 31096.768} C_VEL
LIN {X 0,Y 640.817,Z 620.849,A -85,B 0,C 180,E1 31093.605,E2 31093.605} C_VEL
LIN {X 0,Y 640.757,Z 620.849,A -85,B 0,C 180,E1 31090.819,E2 31090.819} C_VEL
LIN {X 0,Y 640.783,Z 620.847,A -85,B 0,C 180,E1 31087.712,E2 31087.712} C_VEL
LIN {X 0,Y 640.793,Z 620.846,A -85,B 0,C 180,E1 31084.828,E2 31084.828} C_VEL
LIN {X 0,Y 640.815,Z 620.841,A -85,B 0,C 180,E1 31081.62,E2 31081.62} C_VEL
LIN {X 0,Y 640.806,Z 620.846,A -85,B 0,C 180,E1 31078.546,E2 31078.546} C_VEL
LIN {X 0,Y 640.833,Z 620.844,A -85,B 0,C 180,E1 31075.41,E2 31075.41} C_VEL
LIN {X 0,Y 640.746,Z 620.847,A -85,B 0,C 180,E1 31072.479,E2 31072.479} C_VEL
LIN {X 0,Y 640.81,Z 620.844,A -85,B 0,C 180,E1 31069.413,E2 31069.413} C_VEL
LIN {X 0,Y 640.789,Z 620.845,A -85,B 0,C 180,E1 31066.5,E2 31066.5} C_VEL
LIN {X 0,Y 640.83,Z 620.835,A -85,B 0,C 180,E1 31063.353,E2 31063.353} C_VEL
LIN {X 0,Y 640.806,Z 620.844,A -85,B 0,C 180,E1 31060.157,E2 31060.157} C_VEL
LIN {X 0,Y 640.837,Z 620.84,A -85,B 0,C 180,E1 31057.082,E2 31057.082} C_VEL
LIN {X 0,Y 640.745,Z 620.848,A -85,B 0,C 180,E1 31054.118,E2 31054.118} C_VEL
LIN {X 0,Y 640.831,Z 620.845,A -85,B 0,C 180,E1 31051.074,E2 31051.074} C_VEL
LIN {X 0,Y 640.79,Z 620.846,A -85,B 0,C 180,E1 31048.034,E2 31048.034} C_VEL
LIN {X 0,Y 640.829,Z 620.835,A -85,B 0,C 180,E1 31044.899,E2 31044.899} C_VEL
LIN {X 0,Y 640.807,Z 620.845,A -85,B 0,C 180,E1 31041.748,E2 31041.748} C_VEL
LIN {X 0,Y 640.828,Z 620.836,A -85,B 0,C 180,E1 31038.663,E2 31038.663} C_VEL
LIN {X 0,Y 640.744,Z 620.849,A -85,B 0,C 180,E1 31035.702,E2 31035.702} C_VEL
LIN {X 0,Y 640.829,Z 620.846,A -85,B 0,C 180,E1 31032.757,E2 31032.757} C_VEL
LIN {X 0,Y 640.792,Z 620.844,A -85,B 0,C 180,E1 31029.676,E2 31029.676} C_VEL
LIN {X 0,Y 640.82,Z 620.84,A -85,B 0,C 180,E1 31026.653,E2 31026.653} C_VEL
LIN {X 0,Y 640.821,Z 620.848,A -85,B 0,C 180,E1 31023.498,E2 31023.498} C_VEL
LIN {X 0,Y 640.789,Z 620.845,A -85,B 0,C 180,E1 31020.535,E2 31020.535} C_VEL
LIN {X 0,Y 640.753,Z 620.85,A -85,B 0,C 180,E1 31017.417,E2 31017.417} C_VEL
LIN {X 0,Y 640.792,Z 620.849,A -85,B 0,C 180,E1 31014.628,E2 31014.628} C_VEL
LIN {X 0,Y 640.799,Z 620.843,A -85,B 0,C 180,E1 31011.497,E2 31011.497} C_VEL
LIN {X 0,Y 640.817,Z 620.845,A -85,B 0,C 180,E1 31008.463,E2 31008.463} C_VEL
LIN {X 0,Y 640.831,Z 620.845,A -85,B 0,C 180,E1 31005.353,E2 31005.353} C_VEL
LIN {X 0,Y 640.769,Z 620.849,A -85,B 0,C 180,E1 31002.382,E2 31002.382} C_VEL
LIN {X 0,Y 640.786,Z 620.916,A -85,B 0,C 180,E1 30999.945,E2 30999.945} C_VEL
LIN {X 0,Y 645.33,Z 638.222,A -85,B 0,C 180,E1 30998.471,E2 30998.471} C_VEL
LIN {X 0,Y 644.781,Z 684.495,A -85,B 0,C 180,E1 30995.039,E2 30995.039} C_VEL
LIN {X 0,Y 644.263,Z 726.11,A -85,B 0,C 180,E1 30991.95,E2 30991.95} C_VEL
LIN {X 0,Y 643.575,Z 768.586,A -85,B 0,C 180,E1 30988.789,E2 30988.789} C_VEL
LIN {X 0,Y 642.943,Z 810.339,A -85,B 0,C 180,E1 30985.679,E2 30985.679} C_VEL
LIN {X 0,Y 642.84,Z 822.497,A -85,B 0,C 180,E1 30984.814,E2 30984.814} C_VEL
LIN {X 0,Y 643.205,Z 830.053,A -85,B 0,C 180,E1 30984.715,E2 30984.715} C_VEL
LIN {X 0,Y 642.431,Z 964.59,A -85,B 0,C 180,E1 30983.112,E2 30983.112} C_VEL
LIN {X 0,Y 642.305,Z 980.86,A -85,B 0,C 180,E1 30982.748,E2 30982.748} C_VEL
LIN {X 0,Y 642.121,Z 996.476,A -85,B 0,C 180,E1 30982.231,E2 30982.231} C_VEL
LIN {X 0,Y 641.863,Z 1011.221,A -85,B 0,C 180,E1 30981.568,E2 30981.568} C_VEL
LIN {X 0,Y 641.592,Z 1025.848,A -85,B 0,C 180,E1 30980.715,E2 30980.715} C_VEL
LIN {X 0,Y 641.285,Z 1038.523,A -85,B 0,C 180,E1 30979.774,E2 30979.774} C_VEL
LIN {X 0,Y 641.021,Z 1049.759,A -85,B 0,C 180,E1 30978.741,E2 30978.741} C_VEL
LIN {X 0,Y 640.78,Z 1059.565,A -85,B 0,C 180,E1 30977.619,E2 30977.619} C_VEL
LIN {X 0,Y 640.579,Z 1068.589,A -85,B 0,C 180,E1 30976.315,E2 30976.315} C_VEL
LIN {X 0,Y 640.441,Z 1075.485,A -85,B 0,C 180,E1 30975.018,E2 30975.018} C_VEL
LIN {X 0,Y 640.356,Z 1081.198,A -85,B 0,C 180,E1 30973.543,E2 30973.543} C_VEL
LIN {X 0,Y 640.299,Z 1085,A -85,B 0,C 180,E1 30971.985,E2 30971.985} C_VEL
LIN {X 0,Y 640.284,Z 1086.713,A -85,B 0,C 180,E1 30970.526,E2 30970.526} C_VEL
LIN {X 0,Y 640.302,Z 1086.574,A -85,B 0,C 180,E1 30969.072,E2 30969.072} C_VEL
LIN {X 0,Y 640.344,Z 1084.727,A -85,B 0,C 180,E1 30967.625,E2 30967.625} C_VEL
LIN {X 0,Y 640.406,Z 1081.001,A -85,B 0,C 180,E1 30966.183,E2 30966.183} C_VEL
LIN {X 0,Y 640.516,Z 1075.786,A -85,B 0,C 180,E1 30964.834,E2 30964.834} C_VEL
LIN {X 0,Y 640.676,Z 1068.613,A -85,B 0,C 180,E1 30963.488,E2 30963.488} C_VEL
LIN {X 0,Y 640.892,Z 1059.944,A -85,B 0,C 180,E1 30962.233,E2 30962.233} C_VEL
LIN {X 0,Y 641.152,Z 1049.685,A -85,B 0,C 180,E1 30961.07,E2 30961.07} C_VEL
LIN {X 0,Y 641.448,Z 1037.867,A -85,B 0,C 180,E1 30959.998,E2 30959.998} C_VEL
LIN {X 0,Y 641.735,Z 1024.787,A -85,B 0,C 180,E1 30959.061,E2 30959.061} C_VEL
LIN {X 0,Y 641.971,Z 1010.652,A -85,B 0,C 180,E1 30958.258,E2 30958.258} C_VEL
LIN {X 0,Y 642.193,Z 996.087,A -85,B 0,C 180,E1 30957.633,E2 30957.633} C_VEL
LIN {X 0,Y 642.342,Z 982.469,A -85,B 0,C 180,E1 30957.193,E2 30957.193} C_VEL
LIN {X 0,Y 642.431,Z 967.38,A -85,B 0,C 180,E1 30956.842,E2 30956.842} C_VEL
LIN {X 0,Y 642.571,Z 926.994,A -85,B 0,C 180,E1 30956.342,E2 30956.342} C_VEL
LIN {X 0,Y 643.222,Z 824.758,A -85,B 0,C 180,E1 30955.094,E2 30955.094} C_VEL
LIN {X 0,Y 643.762,Z 782.582,A -85,B 0,C 180,E1 30952.008,E2 30952.008} C_VEL
LIN {X 0,Y 644.13,Z 746.042,A -85,B 0,C 180,E1 30949.353,E2 30949.353} C_VEL
LIN {X 0,Y 644.442,Z 706.477,A -85,B 0,C 180,E1 30946.54,E2 30946.54} C_VEL
LIN {X 0,Y 644.383,Z 667.638,A -85,B 0,C 180,E1 30943.835,E2 30943.835} C_VEL
LIN {X 0,Y 644.292,Z 633.863,A -85,B 0,C 180,E1 30941.541,E2 30941.541} C_VEL
LIN {X 0,Y 640.791,Z 620.851,A -85,B 0,C 180,E1 30940.523,E2 30940.523} C_VEL
LIN {X 0,Y 640.829,Z 620.851,A -85,B 0,C 180,E1 30937.33,E2 30937.33} C_VEL
LIN {X 0,Y 640.833,Z 620.848,A -85,B 0,C 180,E1 30934.192,E2 30934.192} C_VEL
LIN {X 0,Y 640.791,Z 620.849,A -85,B 0,C 180,E1 30931.07,E2 30931.07} C_VEL
LIN {X 0,Y 640.8,Z 620.847,A -85,B 0,C 180,E1 30928.168,E2 30928.168} C_VEL
LIN {X 0,Y 640.823,Z 620.846,A -85,B 0,C 180,E1 30924.955,E2 30924.955} C_VEL
LIN {X 0,Y 640.832,Z 620.846,A -85,B 0,C 180,E1 30921.837,E2 30921.837} C_VEL
LIN {X 0,Y 640.796,Z 620.848,A -85,B 0,C 180,E1 30918.77,E2 30918.77} C_VEL
LIN {X 0,Y 640.808,Z 620.847,A -85,B 0,C 180,E1 30915.773,E2 30915.773} C_VEL
LIN {X 0,Y 640.82,Z 620.844,A -85,B 0,C 180,E1 30912.5,E2 30912.5} C_VEL
LIN {X 0,Y 640.834,Z 620.844,A -85,B 0,C 180,E1 30909.421,E2 30909.421} C_VEL
LIN {X 0,Y 640.802,Z 620.85,A -85,B 0,C 180,E1 30906.364,E2 30906.364} C_VEL
LIN {X 0,Y 640.804,Z 620.942,A -85,B 0,C 180,E1 30905.766,E2 30905.766} C_VEL
LIN {X 0,Y 648.441,Z 645.103,A -85,B 0,C 180,E1 30903.187,E2 30903.187} C_VEL
LIN {X 0,Y 649.337,Z 649.268,A -85,B 0,C 180,E1 30902.777,E2 30902.777} C_VEL
LIN {X 0,Y 648.017,Z 681.747,A -85,B 0,C 180,E1 30900.096,E2 30900.096} C_VEL
LIN {X 0,Y 652.758,Z 705.256,A -85,B 0,C 180,E1 30899.539,E2 30899.539} C_VEL
LIN {X 0,Y 651.258,Z 829.707,A -85,B 0,C 180,E1 30898.026,E2 30898.026} C_VEL
LIN {X 0,Y 649.703,Z 982.141,A -85,B 0,C 180,E1 30896.198,E2 30896.198} C_VEL
LIN {X 0,Y 649.163,Z 1005.102,A -85,B 0,C 180,E1 30895.784,E2 30895.784} C_VEL
LIN {X 0,Y 648.493,Z 1026.816,A -85,B 0,C 180,E1 30895.233,E2 30895.233} C_VEL
LIN {X 0,Y 647.702,Z 1047.871,A -85,B 0,C 180,E1 30894.534,E2 30894.534} C_VEL
LIN {X 0,Y 646.811,Z 1068.145,A -85,B 0,C 180,E1 30893.697,E2 30893.697} C_VEL
LIN {X 0,Y 645.868,Z 1088.605,A -85,B 0,C 180,E1 30892.676,E2 30892.676} C_VEL
LIN {X 0,Y 644.922,Z 1107.51,A -85,B 0,C 180,E1 30891.556,E2 30891.556} C_VEL
LIN {X 0,Y 643.987,Z 1125.258,A -85,B 0,C 180,E1 30890.312,E2 30890.312} C_VEL
LIN {X 0,Y 643.079,Z 1142.928,A -85,B 0,C 180,E1 30888.868,E2 30888.868} C_VEL
LIN {X 0,Y 642.341,Z 1157.487,A -85,B 0,C 180,E1 30887.482,E2 30887.482} C_VEL
LIN {X 0,Y 641.625,Z 1171.326,A -85,B 0,C 180,E1 30885.917,E2 30885.917} C_VEL
LIN {X 0,Y 641.023,Z 1184.549,A -85,B 0,C 180,E1 30884.174,E2 30884.174} C_VEL
LIN {X 0,Y 640.596,Z 1195.753,A -85,B 0,C 180,E1 30882.438,E2 30882.438} C_VEL
LIN {X 0,Y 640.29,Z 1205.514,A -85,B 0,C 180,E1 30880.617,E2 30880.617} C_VEL
LIN {X 0,Y 640.086,Z 1213.824,A -85,B 0,C 180,E1 30878.714,E2 30878.714} C_VEL
LIN {X 0,Y 639.967,Z 1220.387,A -85,B 0,C 180,E1 30876.818,E2 30876.818} C_VEL
LIN {X 0,Y 639.916,Z 1225.229,A -85,B 0,C 180,E1 30874.929,E2 30874.929} C_VEL
LIN {X 0,Y 639.904,Z 1228.561,A -85,B 0,C 180,E1 30872.954,E2 30872.954} C_VEL
LIN {X 0,Y 639.905,Z 1230.236,A -85,B 0,C 180,E1 30871.073,E2 30871.073} C_VEL
LIN {X 0,Y 639.91,Z 1230.303,A -85,B 0,C 180,E1 30869.193,E2 30869.193} C_VEL
LIN {X 0,Y 639.911,Z 1228.782,A -85,B 0,C 180,E1 30867.222,E2 30867.222} C_VEL
LIN {X 0,Y 639.92,Z 1225.816,A -85,B 0,C 180,E1 30865.338,E2 30865.338} C_VEL
LIN {X 0,Y 639.962,Z 1221.142,A -85,B 0,C 180,E1 30863.45,E2 30863.45} C_VEL
LIN {X 0,Y 640.08,Z 1214.395,A -85,B 0,C 180,E1 30861.433,E2 30861.433} C_VEL
LIN {X 0,Y 640.264,Z 1206.416,A -85,B 0,C 180,E1 30859.562,E2 30859.562} C_VEL
LIN {X 0,Y 640.552,Z 1196.745,A -85,B 0,C 180,E1 30857.738,E2 30857.738} C_VEL
LIN {X 0,Y 640.995,Z 1185.167,A -85,B 0,C 180,E1 30855.915,E2 30855.915} C_VEL
LIN {X 0,Y 641.564,Z 1172.845,A -85,B 0,C 180,E1 30854.264,E2 30854.264} C_VEL
LIN {X 0,Y 642.249,Z 1159.157,A -85,B 0,C 180,E1 30852.7,E2 30852.7} C_VEL
LIN {X 0,Y 642.966,Z 1144.934,A -85,B 0,C 180,E1 30851.315,E2 30851.315} C_VEL
LIN {X 0,Y 643.762,Z 1129.145,A -85,B 0,C 180,E1 30850.001,E2 30850.001} C_VEL
LIN {X 0,Y 644.643,Z 1111.017,A -85,B 0,C 180,E1 30848.717,E2 30848.717} C_VEL
LIN {X 0,Y 645.541,Z 1091.688,A -85,B 0,C 180,E1 30847.553,E2 30847.553} C_VEL
LIN {X 0,Y 646.411,Z 1072.503,A -85,B 0,C 180,E1 30846.575,E2 30846.575} C_VEL
LIN {X 0,Y 647.24,Z 1051.4,A -85,B 0,C 180,E1 30845.687,E2 30845.687} C_VEL
LIN {X 0,Y 647.973,Z 1030.724,A -85,B 0,C 180,E1 30844.987,E2 30844.987} C_VEL
LIN {X 0,Y 648.606,Z 1008.505,A -85,B 0,C 180,E1 30844.397,E2 30844.397} C_VEL
LIN {X 0,Y 649.163,Z 986.007,A -85,B 0,C 180,E1 30843.967,E2 30843.967} C_VEL
LIN {X 0,Y 651.23,Z 784.682,A -85,B 0,C 180,E1 30841.531,E2 30841.531} C_VEL
LIN {X 0,Y 652.354,Z 703.313,A -85,B 0,C 180,E1 30840.463,E2 30840.463} C_VEL
LIN {X 0,Y 647.407,Z 677.716,A -85,B 0,C 180,E1 30839.802,E2 30839.802} C_VEL
LIN {X 0,Y 648.676,Z 647.088,A -85,B 0,C 180,E1 30837.245,E2 30837.245} C_VEL
LIN {X 0,Y 643.794,Z 630.086,A -85,B 0,C 180,E1 30835.403,E2 30835.403} C_VEL
LIN {X 0,Y 640.827,Z 620.848,A -85,B 0,C 180,E1 30834.298,E2 30834.298} C_VEL
LIN {X 0,Y 640.815,Z 620.845,A -85,B 0,C 180,E1 30831.135,E2 30831.135} C_VEL
LIN {X 0,Y 640.808,Z 620.85,A -85,B 0,C 180,E1 30827.859,E2 30827.859} C_VEL
LIN {X 0,Y 640.826,Z 620.844,A -85,B 0,C 180,E1 30824.769,E2 30824.769} C_VEL
LIN {X 0,Y 640.791,Z 620.85,A -85,B 0,C 180,E1 30821.631,E2 30821.631} C_VEL
LIN {X 0,Y 640.826,Z 620.845,A -85,B 0,C 180,E1 30818.619,E2 30818.619} C_VEL
LIN {X 0,Y 640.781,Z 620.851,A -85,B 0,C 180,E1 30815.457,E2 30815.457} C_VEL
LIN {X 0,Y 640.809,Z 620.849,A -85,B 0,C 180,E1 30812.571,E2 30812.571} C_VEL
LIN {X 0,Y 640.805,Z 620.985,A -85,B 0,C 180,E1 30811.598,E2 30811.598} C_VEL
LIN {X 0,Y 643.872,Z 630.413,A -85,B 0,C 180,E1 30810.295,E2 30810.295} C_VEL
LIN {X 0,Y 652.503,Z 647.131,A -85,B 0,C 180,E1 30809.55,E2 30809.55} C_VEL
LIN {X 0,Y 653.01,Z 649.073,A -85,B 0,C 180,E1 30809.496,E2 30809.496} C_VEL
LIN {X 0,Y 650.877,Z 781.18,A -85,B 0,C 180,E1 30807.784,E2 30807.784} C_VEL
LIN {X 0,Y 649.332,Z 930.213,A -85,B 0,C 180,E1 30805.978,E2 30805.978} C_VEL
LIN {X 0,Y 648.833,Z 952.488,A -85,B 0,C 180,E1 30805.542,E2 30805.542} C_VEL
LIN {X 0,Y 648.229,Z 973.37,A -85,B 0,C 180,E1 30804.979,E2 30804.979} C_VEL
LIN {X 0,Y 647.531,Z 993.169,A -85,B 0,C 180,E1 30804.302,E2 30804.302} C_VEL
LIN {X 0,Y 646.704,Z 1012.873,A -85,B 0,C 180,E1 30803.463,E2 30803.463} C_VEL
LIN {X 0,Y 645.807,Z 1031.918,A -85,B 0,C 180,E1 30802.486,E2 30802.486} C_VEL
LIN {X 0,Y 644.85,Z 1050.932,A -85,B 0,C 180,E1 30801.324,E2 30801.324} C_VEL
LIN {X 0,Y 643.919,Z 1068.332,A -85,B 0,C 180,E1 30800.072,E2 30800.072} C_VEL
LIN {X 0,Y 642.998,Z 1085.216,A -85,B 0,C 180,E1 30798.638,E2 30798.638} C_VEL
LIN {X 0,Y 642.224,Z 1099.566,A -85,B 0,C 180,E1 30797.208,E2 30797.208} C_VEL
LIN {X 0,Y 641.504,Z 1113.931,A -85,B 0,C 180,E1 30795.552,E2 30795.552} C_VEL
LIN {X 0,Y 640.956,Z 1126.162,A -85,B 0,C 180,E1 30793.902,E2 30793.902} C_VEL
LIN {X 0,Y 640.549,Z 1137.013,A -85,B 0,C 180,E1 30792.167,E2 30792.167} C_VEL
LIN {X 0,Y 640.245,Z 1146.836,A -85,B 0,C 180,E1 30790.297,E2 30790.297} C_VEL
LIN {X 0,Y 640.062,Z 1154.72,A -85,B 0,C 180,E1 30788.446,E2 30788.446} C_VEL
LIN {X 0,Y 639.961,Z 1161.01,A -85,B 0,C 180,E1 30786.551,E2 30786.551} C_VEL
LIN {X 0,Y 639.923,Z 1165.718,A -85,B 0,C 180,E1 30784.662,E2 30784.662} C_VEL
LIN {X 0,Y 639.915,Z 1168.727,A -85,B 0,C 180,E1 30782.778,E2 30782.778} C_VEL
LIN {X 0,Y 639.91,Z 1170.312,A -85,B 0,C 180,E1 30780.718,E2 30780.718} C_VEL
LIN {X 0,Y 639.91,Z 1170.221,A -85,B 0,C 180,E1 30778.838,E2 30778.838} C_VEL
LIN {X 0,Y 639.92,Z 1168.389,A -85,B 0,C 180,E1 30776.867,E2 30776.867} C_VEL
LIN {X 0,Y 639.936,Z 1164.934,A -85,B 0,C 180,E1 30774.892,E2 30774.892} C_VEL
LIN {X 0,Y 639.984,Z 1159.985,A -85,B 0,C 180,E1 30773.002,E2 30773.002} C_VEL
LIN {X 0,Y 640.09,Z 1153.295,A -85,B 0,C 180,E1 30771.106,E2 30771.106} C_VEL
LIN {X 0,Y 640.29,Z 1145.321,A -85,B 0,C 180,E1 30769.293,E2 30769.293} C_VEL
LIN {X 0,Y 640.582,Z 1135.978,A -85,B 0,C 180,E1 30767.563,E2 30767.563} C_VEL
LIN {X 0,Y 641.04,Z 1124.229,A -85,B 0,C 180,E1 30765.735,E2 30765.735} C_VEL
LIN {X 0,Y 641.63,Z 1111.504,A -85,B 0,C 180,E1 30764.052,E2 30764.052} C_VEL
LIN {X 0,Y 642.354,Z 1096.97,A -85,B 0,C 180,E1 30762.426,E2 30762.426} C_VEL
LIN {X 0,Y 643.195,Z 1081.507,A -85,B 0,C 180,E1 30760.941,E2 30760.941} C_VEL
LIN {X 0,Y 644.124,Z 1064.75,A -85,B 0,C 180,E1 30759.56,E2 30759.56} C_VEL
LIN {X 0,Y 645.102,Z 1047.04,A -85,B 0,C 180,E1 30758.313,E2 30758.313} C_VEL
LIN {X 0,Y 646.089,Z 1028.161,A -85,B 0,C 180,E1 30757.193,E2 30757.193} C_VEL
LIN {X 0,Y 647.04,Z 1007.874,A -85,B 0,C 180,E1 30756.183,E2 30756.183} C_VEL
LIN {X 0,Y 647.987,Z 986.356,A -85,B 0,C 180,E1 30755.31,E2 30755.31} C_VEL
LIN {X 0,Y 648.764,Z 964.986,A -85,B 0,C 180,E1 30754.621,E2 30754.621} C_VEL
LIN {X 0,Y 649.411,Z 943.103,A -85,B 0,C 180,E1 30754.088,E2 30754.088} C_VEL
LIN {X 0,Y 649.847,Z 920.712,A -85,B 0,C 180,E1 30753.712,E2 30753.712} C_VEL
LIN {X 0,Y 651.118,Z 798.959,A -85,B 0,C 180,E1 30752.259,E2 30752.259} C_VEL
LIN {X 0,Y 650.349,Z 791.377,A -85,B 0,C 180,E1 30752.129,E2 30752.129} C_VEL
LIN {X 0,Y 644.976,Z 771.584,A -85,B 0,C 180,E1 30751.635,E2 30751.635} C_VEL
LIN {X 0,Y 644.381,Z 765.068,A -85,B 0,C 180,E1 30751.524,E2 30751.524} C_VEL
LIN {X 0,Y 645.841,Z 650.31,A -85,B 0,C 180,E1 30750.078,E2 30750.078} C_VEL
LIN {X 0,Y 635.42,Z 629.199,A -85,B 0,C 180,E1 30749.245,E2 30749.245} C_VEL
LIN {X 0,Y 634.061,Z 626.219,A -85,B 0,C 180,E1 30749.123,E2 30749.123} C_VEL
LIN {X 0,Y 632.888,Z 621.838,A -85,B 0,C 180,E1 30748.555,E2 30748.555} C_VEL
LIN {X 0,Y 632.814,Z 621.842,A -85,B 0,C 180,E1 30745.555,E2 30745.555} C_VEL
LIN {X 0,Y 632.891,Z 621.83,A -85,B 0,C 180,E1 30742.477,E2 30742.477} C_VEL
LIN {X 0,Y 632.89,Z 621.837,A -85,B 0,C 180,E1 30739.274,E2 30739.274} C_VEL
LIN {X 0,Y 632.891,Z 621.829,A -85,B 0,C 180,E1 30736.09,E2 30736.09} C_VEL
LIN {X 0,Y 632.836,Z 621.836,A -85,B 0,C 180,E1 30733.045,E2 30733.045} C_VEL
LIN {X 0,Y 632.885,Z 621.835,A -85,B 0,C 180,E1 30730.018,E2 30730.018} C_VEL
LIN {X 0,Y 632.822,Z 621.837,A -85,B 0,C 180,E1 30727.014,E2 30727.014} C_VEL
LIN {X 0,Y 632.891,Z 621.83,A -85,B 0,C 180,E1 30723.965,E2 30723.965} C_VEL
LIN {X 0,Y 632.893,Z 621.836,A -85,B 0,C 180,E1 30720.751,E2 30720.751} C_VEL
LIN {X 0,Y 632.894,Z 621.831,A -85,B 0,C 180,E1 30717.575,E2 30717.575} C_VEL
LIN {X 0,Y 632.833,Z 621.837,A -85,B 0,C 180,E1 30714.555,E2 30714.555} C_VEL
LIN {X 0,Y 632.884,Z 621.835,A -85,B 0,C 180,E1 30711.6,E2 30711.6} C_VEL
LIN {X 0,Y 632.826,Z 621.835,A -85,B 0,C 180,E1 30708.564,E2 30708.564} C_VEL
LIN {X 0,Y 632.896,Z 621.828,A -85,B 0,C 180,E1 30705.487,E2 30705.487} C_VEL
LIN {X 0,Y 632.889,Z 621.834,A -85,B 0,C 180,E1 30702.316,E2 30702.316} C_VEL
LIN {X 0,Y 632.893,Z 621.828,A -85,B 0,C 180,E1 30699.091,E2 30699.091} C_VEL
LIN {X 0,Y 632.825,Z 621.837,A -85,B 0,C 180,E1 30696.078,E2 30696.078} C_VEL
LIN {X 0,Y 632.874,Z 621.832,A -85,B 0,C 180,E1 30693.08,E2 30693.08} C_VEL
LIN {X 0,Y 632.831,Z 621.835,A -85,B 0,C 180,E1 30690.092,E2 30690.092} C_VEL
LIN {X 0,Y 632.89,Z 621.824,A -85,B 0,C 180,E1 30687.013,E2 30687.013} C_VEL
LIN {X 0,Y 632.889,Z 621.835,A -85,B 0,C 180,E1 30683.834,E2 30683.834} C_VEL
LIN {X 0,Y 632.894,Z 621.829,A -85,B 0,C 180,E1 30680.636,E2 30680.636} C_VEL
LIN {X 0,Y 632.82,Z 621.832,A -85,B 0,C 180,E1 30677.593,E2 30677.593} C_VEL
LIN {X 0,Y 632.886,Z 621.837,A -85,B 0,C 180,E1 30674.61,E2 30674.61} C_VEL
LIN {X 0,Y 632.838,Z 621.835,A -85,B 0,C 180,E1 30671.58,E2 30671.58} C_VEL
LIN {X 0,Y 632.892,Z 621.829,A -85,B 0,C 180,E1 30668.5,E2 30668.5} C_VEL
LIN {X 0,Y 632.882,Z 621.835,A -85,B 0,C 180,E1 30665.251,E2 30665.251} C_VEL
LIN {X 0,Y 632.896,Z 621.831,A -85,B 0,C 180,E1 30662.121,E2 30662.121} C_VEL
LIN {X 0,Y 632.818,Z 621.838,A -85,B 0,C 180,E1 30659.209,E2 30659.209} C_VEL
LIN {X 0,Y 632.88,Z 621.838,A -85,B 0,C 180,E1 30656.199,E2 30656.199} C_VEL
LIN {X 0,Y 632.843,Z 621.835,A -85,B 0,C 180,E1 30653.104,E2 30653.104} C_VEL
LIN {X 0,Y 632.894,Z 621.829,A -85,B 0,C 180,E1 30649.986,E2 30649.986} C_VEL
LIN {X 0,Y 632.877,Z 621.835,A -85,B 0,C 180,E1 30646.743,E2 30646.743} C_VEL
LIN {X 0,Y 632.893,Z 621.833,A -85,B 0,C 180,E1 30643.652,E2 30643.652} C_VEL
LIN {X 0,Y 632.81,Z 621.843,A -85,B 0,C 180,E1 30640.676,E2 30640.676} C_VEL
LIN {X 0,Y 632.818,Z 621.85,A -85,B 0,C 180,E1 30640.189,E2 30640.189} C_VEL
LIN {X 0,Y 637.727,Z 641.124,A -85,B 0,C 180,E1 30638.55,E2 30638.55} C_VEL
LIN {X 0,Y 637.124,Z 686.614,A -85,B 0,C 180,E1 30635.154,E2 30635.154} C_VEL
LIN {X 0,Y 636.566,Z 728.041,A -85,B 0,C 180,E1 30632.064,E2 30632.064} C_VEL
LIN {X 0,Y 635.867,Z 769.956,A -85,B 0,C 180,E1 30628.937,E2 30628.937} C_VEL
LIN {X 0,Y 635.198,Z 811.977,A -85,B 0,C 180,E1 30625.793,E2 30625.793} C_VEL
LIN {X 0,Y 635.083,Z 823.15,A -85,B 0,C 180,E1 30624.989,E2 30624.989} C_VEL
LIN {X 0,Y 635.453,Z 830.62,A -85,B 0,C 180,E1 30624.888,E2 30624.888} C_VEL
LIN {X 0,Y 634.614,Z 965.364,A -85,B 0,C 180,E1 30623.255,E2 30623.255} C_VEL
LIN {X 0,Y 634.49,Z 981.541,A -85,B 0,C 180,E1 30622.89,E2 30622.89} C_VEL
LIN {X 0,Y 634.299,Z 997.016,A -85,B 0,C 180,E1 30622.374,E2 30622.374} C_VEL
LIN {X 0,Y 634.03,Z 1011.862,A -85,B 0,C 180,E1 30621.702,E2 30621.702} C_VEL
LIN {X 0,Y 633.74,Z 1026.614,A -85,B 0,C 180,E1 30620.835,E2 30620.835} C_VEL
LIN {X 0,Y 633.417,Z 1039.275,A -85,B 0,C 180,E1 30619.885,E2 30619.885} C_VEL
LIN {X 0,Y 633.126,Z 1051.026,A -85,B 0,C 180,E1 30618.792,E2 30618.792} C_VEL
LIN {X 0,Y 632.847,Z 1061.465,A -85,B 0,C 180,E1 30617.562,E2 30617.562} C_VEL
LIN {X 0,Y 632.655,Z 1069.748,A -85,B 0,C 180,E1 30616.337,E2 30616.337} C_VEL
LIN {X 0,Y 632.505,Z 1076.616,A -85,B 0,C 180,E1 30615.016,E2 30615.016} C_VEL
LIN {X 0,Y 632.417,Z 1082.267,A -85,B 0,C 180,E1 30613.53,E2 30613.53} C_VEL
LIN {X 0,Y 632.353,Z 1086.014,A -85,B 0,C 180,E1 30611.953,E2 30611.953} C_VEL
LIN {X 0,Y 632.338,Z 1087.666,A -85,B 0,C 180,E1 30610.475,E2 30610.475} C_VEL
LIN {X 0,Y 632.364,Z 1087.425,A -85,B 0,C 180,E1 30608.912,E2 30608.912} C_VEL
LIN {X 0,Y 632.408,Z 1085.372,A -85,B 0,C 180,E1 30607.447,E2 30607.447} C_VEL
LIN {X 0,Y 632.49,Z 1081.481,A -85,B 0,C 180,E1 30605.987,E2 30605.987} C_VEL
LIN {X 0,Y 632.62,Z 1076.043,A -85,B 0,C 180,E1 30604.621,E2 30604.621} C_VEL
LIN {X 0,Y 632.802,Z 1068.64,A -85,B 0,C 180,E1 30603.259,E2 30603.259} C_VEL
LIN {X 0,Y 633.022,Z 1060.407,A -85,B 0,C 180,E1 30602.08,E2 30602.08} C_VEL
LIN {X 0,Y 633.307,Z 1049.988,A -85,B 0,C 180,E1 30600.903,E2 30600.903} C_VEL
LIN {X 0,Y 633.614,Z 1038.544,A -85,B 0,C 180,E1 30599.862,E2 30599.862} C_VEL
LIN {X 0,Y 633.919,Z 1025.391,A -85,B 0,C 180,E1 30598.914,E2 30598.914} C_VEL
LIN {X 0,Y 634.159,Z 1012.051,A -85,B 0,C 180,E1 30598.146,E2 30598.146} C_VEL
LIN {X 0,Y 634.393,Z 997.665,A -85,B 0,C 180,E1 30597.514,E2 30597.514} C_VEL
LIN {X 0,Y 634.556,Z 983.627,A -85,B 0,C 180,E1 30597.051,E2 30597.051} C_VEL
LIN {X 0,Y 634.646,Z 968.502,A -85,B 0,C 180,E1 30596.693,E2 30596.693} C_VEL
LIN {X 0,Y 634.767,Z 932.398,A -85,B 0,C 180,E1 30596.236,E2 30596.236} C_VEL
LIN {X 0,Y 635.539,Z 825.91,A -85,B 0,C 180,E1 30594.921,E2 30594.921} C_VEL
LIN {X 0,Y 636.143,Z 783.222,A -85,B 0,C 180,E1 30591.775,E2 30591.775} C_VEL
LIN {X 0,Y 636.501,Z 747.446,A -85,B 0,C 180,E1 30589.178,E2 30589.178} C_VEL
LIN {X 0,Y 636.839,Z 710.856,A -85,B 0,C 180,E1 30586.562,E2 30586.562} C_VEL
LIN {X 0,Y 636.845,Z 670.368,A -85,B 0,C 180,E1 30583.723,E2 30583.723} C_VEL
LIN {X 0,Y 636.852,Z 636.446,A -85,B 0,C 180,E1 30581.413,E2 30581.413} C_VEL
LIN {X 0,Y 632.862,Z 621.839,A -85,B 0,C 180,E1 30580.273,E2 30580.273} C_VEL
LIN {X 0,Y 632.891,Z 621.84,A -85,B 0,C 180,E1 30577.128,E2 30577.128} C_VEL
LIN {X 0,Y 632.894,Z 621.834,A -85,B 0,C 180,E1 30573.845,E2 30573.845} C_VEL
LIN {X 0,Y 632.854,Z 621.839,A -85,B 0,C 180,E1 30570.672,E2 30570.672} C_VEL
LIN {X 0,Y 632.891,Z 621.835,A -85,B 0,C 180,E1 30567.615,E2 30567.615} C_VEL
LIN {X 0,Y 632.882,Z 621.838,A -85,B 0,C 180,E1 30564.56,E2 30564.56} C_VEL
LIN {X 0,Y 632.888,Z 621.833,A -85,B 0,C 180,E1 30561.27,E2 30561.27} C_VEL
LIN {X 0,Y 632.856,Z 621.837,A -85,B 0,C 180,E1 30558.182,E2 30558.182} C_VEL
LIN {X 0,Y 632.893,Z 621.834,A -85,B 0,C 180,E1 30555.052,E2 30555.052} C_VEL
LIN {X 0,Y 632.876,Z 621.837,A -85,B 0,C 180,E1 30551.913,E2 30551.913} C_VEL
LIN {X 0,Y 632.874,Z 621.835,A -85,B 0,C 180,E1 30548.611,E2 30548.611} C_VEL
LIN {X 0,Y 632.862,Z 621.913,A -85,B 0,C 180,E1 30546.16,E2 30546.16} C_VEL
LIN {X 0,Y 640.733,Z 646.642,A -85,B 0,C 180,E1 30543.475,E2 30543.475} C_VEL
LIN {X 0,Y 641.991,Z 651.511,A -85,B 0,C 180,E1 30542.978,E2 30542.978} C_VEL
LIN {X 0,Y 640.663,Z 681.425,A -85,B 0,C 180,E1 30540.478,E2 30540.478} C_VEL
LIN {X 0,Y 645.756,Z 706.686,A -85,B 0,C 180,E1 30539.868,E2 30539.868} C_VEL
LIN {X 0,Y 643.816,Z 850.046,A -85,B 0,C 180,E1 30538.087,E2 30538.087} C_VEL
LIN {X 0,Y 642.373,Z 980.998,A -85,B 0,C 180,E1 30536.497,E2 30536.497} C_VEL
LIN {X 0,Y 641.799,Z 1004.224,A -85,B 0,C 180,E1 30536.079,E2 30536.079} C_VEL
LIN {X 0,Y 641.076,Z 1025.919,A -85,B 0,C 180,E1 30535.527,E2 30535.527} C_VEL
LIN {X 0,Y 640.246,Z 1046.534,A -85,B 0,C 180,E1 30534.839,E2 30534.839} C_VEL
LIN {X 0,Y 639.295,Z 1067.012,A -85,B 0,C 180,E1 30533.993,E2 30533.993} C_VEL
LIN {X 0,Y 638.323,Z 1086.85,A -85,B 0,C 180,E1 30533.004,E2 30533.004} C_VEL
LIN {X 0,Y 637.295,Z 1105.646,A -85,B 0,C 180,E1 30531.888,E2 30531.888} C_VEL
LIN {X 0,Y 636.332,Z 1123.296,A -85,B 0,C 180,E1 30530.655,E2 30530.655} C_VEL
LIN {X 0,Y 635.402,Z 1140.108,A -85,B 0,C 180,E1 30529.295,E2 30529.295} C_VEL
LIN {X 0,Y 634.543,Z 1155.979,A -85,B 0,C 180,E1 30527.799,E2 30527.799} C_VEL
LIN {X 0,Y 633.806,Z 1170.351,A -85,B 0,C 180,E1 30526.213,E2 30526.213} C_VEL
LIN {X 0,Y 633.226,Z 1182.643,A -85,B 0,C 180,E1 30524.633,E2 30524.633} C_VEL
LIN {X 0,Y 632.73,Z 1194.107,A -85,B 0,C 180,E1 30522.873,E2 30522.873} C_VEL
LIN {X 0,Y 632.359,Z 1204.137,A -85,B 0,C 180,E1 30521.029,E2 30521.029} C_VEL
LIN {X 0,Y 632.131,Z 1212.765,A -85,B 0,C 180,E1 30519.1,E2 30519.1} C_VEL
LIN {X 0,Y 632.003,Z 1219.321,A -85,B 0,C 180,E1 30517.258,E2 30517.258} C_VEL
LIN {X 0,Y 631.935,Z 1224.402,A -85,B 0,C 180,E1 30515.355,E2 30515.355} C_VEL
LIN {X 0,Y 631.911,Z 1227.992,A -85,B 0,C 180,E1 30513.446,E2 30513.446} C_VEL
LIN {X 0,Y 631.902,Z 1229.951,A -85,B 0,C 180,E1 30511.54,E2 30511.54} C_VEL
LIN {X 0,Y 631.901,Z 1230.393,A -85,B 0,C 180,E1 30509.545,E2 30509.545} C_VEL
LIN {X 0,Y 631.913,Z 1229.332,A -85,B 0,C 180,E1 30507.641,E2 30507.641} C_VEL
LIN {X 0,Y 631.927,Z 1226.614,A -85,B 0,C 180,E1 30505.734,E2 30505.734} C_VEL
LIN {X 0,Y 631.966,Z 1221.903,A -85,B 0,C 180,E1 30503.64,E2 30503.64} C_VEL
LIN {X 0,Y 632.071,Z 1215.93,A -85,B 0,C 180,E1 30501.722,E2 30501.722} C_VEL
LIN {X 0,Y 632.247,Z 1208.062,A -85,B 0,C 180,E1 30499.796,E2 30499.796} C_VEL
LIN {X 0,Y 632.537,Z 1198.824,A -85,B 0,C 180,E1 30497.955,E2 30497.955} C_VEL
LIN {X 0,Y 632.97,Z 1188.339,A -85,B 0,C 180,E1 30496.199,E2 30496.199} C_VEL
LIN {X 0,Y 633.491,Z 1177.108,A -85,B 0,C 180,E1 30494.622,E2 30494.622} C_VEL
LIN {X 0,Y 634.12,Z 1163.721,A -85,B 0,C 180,E1 30493.039,E2 30493.039} C_VEL
LIN {X 0,Y 634.904,Z 1148.492,A -85,B 0,C 180,E1 30491.497,E2 30491.497} C_VEL
LIN {X 0,Y 635.777,Z 1131.627,A -85,B 0,C 180,E1 30490.044,E2 30490.044} C_VEL
LIN {X 0,Y 636.729,Z 1113.071,A -85,B 0,C 180,E1 30488.681,E2 30488.681} C_VEL
LIN {X 0,Y 637.671,Z 1094.234,A -85,B 0,C 180,E1 30487.504,E2 30487.504} C_VEL
LIN {X 0,Y 638.617,Z 1074.523,A -85,B 0,C 180,E1 30486.467,E2 30486.467} C_VEL
LIN {X 0,Y 639.482,Z 1053.898,A -85,B 0,C 180,E1 30485.57,E2 30485.57} C_VEL
LIN {X 0,Y 640.319,Z 1032.306,A -85,B 0,C 180,E1 30484.807,E2 30484.807} C_VEL
LIN {X 0,Y 641.01,Z 1010.465,A -85,B 0,C 180,E1 30484.201,E2 30484.201} C_VEL
LIN {X 0,Y 641.598,Z 988.125,A -85,B 0,C 180,E1 30483.757,E2 30483.757} C_VEL
LIN {X 0,Y 642.031,Z 954.469,A -85,B 0,C 180,E1 30483.322,E2 30483.322} C_VEL
LIN {X 0,Y 643.615,Z 811.644,A -85,B 0,C 180,E1 30481.566,E2 30481.566} C_VEL
LIN {X 0,Y 645.495,Z 705.323,A -85,B 0,C 180,E1 30480.144,E2 30480.144} C_VEL
LIN {X 0,Y 640.054,Z 676.859,A -85,B 0,C 180,E1 30479.384,E2 30479.384} C_VEL
LIN {X 0,Y 641.351,Z 649.927,A -85,B 0,C 180,E1 30477.084,E2 30477.084} C_VEL
LIN {X 0,Y 636.706,Z 633.386,A -85,B 0,C 180,E1 30475.245,E2 30475.245} C_VEL
LIN {X 0,Y 632.867,Z 621.838,A -85,B 0,C 180,E1 30473.779,E2 30473.779} C_VEL
LIN {X 0,Y 632.888,Z 621.834,A -85,B 0,C 180,E1 30470.688,E2 30470.688} C_VEL
LIN {X 0,Y 632.856,Z 621.838,A -85,B 0,C 180,E1 30467.573,E2 30467.573} C_VEL
LIN {X 0,Y 632.893,Z 621.834,A -85,B 0,C 180,E1 30464.546,E2 30464.546} C_VEL
LIN {X 0,Y 632.848,Z 621.839,A -85,B 0,C 180,E1 30461.455,E2 30461.455} C_VEL
LIN {X 0,Y 632.896,Z 621.834,A -85,B 0,C 180,E1 30458.407,E2 30458.407} C_VEL
LIN {X 0,Y 632.837,Z 621.839,A -85,B 0,C 180,E1 30455.331,E2 30455.331} C_VEL
LIN {X 0,Y 632.895,Z 621.835,A -85,B 0,C 180,E1 30452.277,E2 30452.277} C_VEL
LIN {X 0,Y 632.915,Z 621.965,A -85,B 0,C 180,E1 30452.136,E2 30452.136} C_VEL
LIN {X 0,Y 636.022,Z 631.488,A -85,B 0,C 180,E1 30450.756,E2 30450.756} C_VEL
LIN {X 0,Y 644.964,Z 648.234,A -85,B 0,C 180,E1 30449.946,E2 30449.946} C_VEL
LIN {X 0,Y 646.105,Z 651.188,A -85,B 0,C 180,E1 30449.833,E2 30449.833} C_VEL
LIN {X 0,Y 643.633,Z 782.671,A -85,B 0,C 180,E1 30448.071,E2 30448.071} C_VEL
LIN {X 0,Y 641.873,Z 930.982,A -85,B 0,C 180,E1 30446.228,E2 30446.228} C_VEL
LIN {X 0,Y 641.352,Z 953.271,A -85,B 0,C 180,E1 30445.785,E2 30445.785} C_VEL
LIN {X 0,Y 640.693,Z 974.76,A -85,B 0,C 180,E1 30445.194,E2 30445.194} C_VEL
LIN {X 0,Y 639.91,Z 995.548,A -85,B 0,C 180,E1 30444.463,E2 30444.463} C_VEL
LIN {X 0,Y 639.065,Z 1015.07,A -85,B 0,C 180,E1 30443.614,E2 30443.614} C_VEL
LIN {X 0,Y 638.136,Z 1033.464,A -85,B 0,C 180,E1 30442.646,E2 30442.646} C_VEL
LIN {X 0,Y 637.117,Z 1052.644,A -85,B 0,C 180,E1 30441.45,E2 30441.45} C_VEL
LIN {X 0,Y 636.15,Z 1069.821,A -85,B 0,C 180,E1 30440.189,E2 30440.189} C_VEL
LIN {X 0,Y 635.219,Z 1085.937,A -85,B 0,C 180,E1 30438.797,E2 30438.797} C_VEL
LIN {X 0,Y 634.393,Z 1100.462,A -85,B 0,C 180,E1 30437.333,E2 30437.333} C_VEL
LIN {X 0,Y 633.62,Z 1114.686,A -85,B 0,C 180,E1 30435.657,E2 30435.657} C_VEL
LIN {X 0,Y 633.005,Z 1127.427,A -85,B 0,C 180,E1 30433.894,E2 30433.894} C_VEL
LIN {X 0,Y 632.574,Z 1138.064,A -85,B 0,C 180,E1 30432.137,E2 30432.137} C_VEL
LIN {X 0,Y 632.253,Z 1147.843,A -85,B 0,C 180,E1 30430.204,E2 30430.204} C_VEL
LIN {X 0,Y 632.067,Z 1155.432,A -85,B 0,C 180,E1 30428.37,E2 30428.37} C_VEL
LIN {X 0,Y 631.964,Z 1161.527,A -85,B 0,C 180,E1 30426.452,E2 30426.452} C_VEL
LIN {X 0,Y 631.924,Z 1166.205,A -85,B 0,C 180,E1 30424.449,E2 30424.449} C_VEL
LIN {X 0,Y 631.909,Z 1169.073,A -85,B 0,C 180,E1 30422.541,E2 30422.541} C_VEL
LIN {X 0,Y 631.905,Z 1170.334,A -85,B 0,C 180,E1 30420.637,E2 30420.637} C_VEL
LIN {X 0,Y 631.907,Z 1170.187,A -85,B 0,C 180,E1 30418.733,E2 30418.733} C_VEL
LIN {X 0,Y 631.918,Z 1168.352,A -85,B 0,C 180,E1 30416.8,E2 30416.8} C_VEL
LIN {X 0,Y 631.942,Z 1164.721,A -85,B 0,C 180,E1 30414.737,E2 30414.737} C_VEL
LIN {X 0,Y 631.999,Z 1159.722,A -85,B 0,C 180,E1 30412.822,E2 30412.822} C_VEL
LIN {X 0,Y 632.128,Z 1152.93,A -85,B 0,C 180,E1 30410.901,E2 30410.901} C_VEL
LIN {X 0,Y 632.358,Z 1144.384,A -85,B 0,C 180,E1 30408.972,E2 30408.972} C_VEL
LIN {X 0,Y 632.703,Z 1134.704,A -85,B 0,C 180,E1 30407.182,E2 30407.182} C_VEL
LIN {X 0,Y 633.18,Z 1123.572,A -85,B 0,C 180,E1 30405.461,E2 30405.461} C_VEL
LIN {X 0,Y 633.82,Z 1111.005,A -85,B 0,C 180,E1 30403.788,E2 30403.788} C_VEL
LIN {X 0,Y 634.58,Z 1096.985,A -85,B 0,C 180,E1 30402.203,E2 30402.203} C_VEL
LIN {X 0,Y 635.476,Z 1081.522,A -85,B 0,C 180,E1 30400.708,E2 30400.708} C_VEL
LIN {X 0,Y 636.521,Z 1063.959,A -85,B 0,C 180,E1 30399.256,E2 30399.256} C_VEL
LIN {X 0,Y 637.595,Z 1045.221,A -85,B 0,C 180,E1 30397.945,E2 30397.945} C_VEL
LIN {X 0,Y 638.676,Z 1026.13,A -85,B 0,C 180,E1 30396.815,E2 30396.815} C_VEL
LIN {X 0,Y 639.669,Z 1006.021,A -85,B 0,C 180,E1 30395.827,E2 30395.827} C_VEL
LIN {X 0,Y 640.626,Z 984.918,A -85,B 0,C 180,E1 30394.98,E2 30394.98} C_VEL
LIN {X 0,Y 641.479,Z 962.419,A -85,B 0,C 180,E1 30394.268,E2 30394.268} C_VEL
LIN {X 0,Y 642.139,Z 940.784,A -85,B 0,C 180,E1 30393.752,E2 30393.752} C_VEL
LIN {X 0,Y 642.589,Z 918.389,A -85,B 0,C 180,E1 30393.389,E2 30393.389} C_VEL
LIN {X 0,Y 644.381,Z 765.068,A -85,B 0,C 180,E1 30391.524,E2 30391.524} C_VEL
LIN {X 0,Y 643.59,Z 757.492,A -85,B 0,C 180,E1 30391.388,E2 30391.388} C_VEL
LIN {X 0,Y 638.307,Z 737.707,A -85,B 0,C 180,E1 30390.881,E2 30390.881} C_VEL
LIN {X 0,Y 637.752,Z 731.192,A -85,B 0,C 180,E1 30390.768,E2 30390.768} C_VEL
LIN {X 0,Y 638.863,Z 652.766,A -85,B 0,C 180,E1 30389.751,E2 30389.751} C_VEL
LIN {X 0,Y 627.541,Z 629.926,A -85,B 0,C 180,E1 30388.83,E2 30388.83} C_VEL
LIN {X 0,Y 625.916,Z 626.485,A -85,B 0,C 180,E1 30388.678,E2 30388.678} C_VEL
LIN {X 0,Y 624.908,Z 622.832,A -85,B 0,C 180,E1 30388.21,E2 30388.21} C_VEL
LIN {X 0,Y 624.889,Z 622.829,A -85,B 0,C 180,E1 30385.278,E2 30385.278} C_VEL
LIN {X 0,Y 624.921,Z 622.821,A -85,B 0,C 180,E1 30382.075,E2 30382.075} C_VEL
LIN {X 0,Y 624.946,Z 622.822,A -85,B 0,C 180,E1 30379.009,E2 30379.009} C_VEL
LIN {X 0,Y 624.951,Z 622.822,A -85,B 0,C 180,E1 30375.79,E2 30375.79} C_VEL
LIN {X 0,Y 624.902,Z 622.824,A -85,B 0,C 180,E1 30372.745,E2 30372.745} C_VEL
LIN {X 0,Y 624.885,Z 622.829,A -85,B 0,C 180,E1 30369.538,E2 30369.538} C_VEL
LIN {X 0,Y 624.901,Z 622.826,A -85,B 0,C 180,E1 30366.718,E2 30366.718} C_VEL
LIN {X 0,Y 624.924,Z 622.821,A -85,B 0,C 180,E1 30363.506,E2 30363.506} C_VEL
LIN {X 0,Y 624.939,Z 622.821,A -85,B 0,C 180,E1 30360.42,E2 30360.42} C_VEL
LIN {X 0,Y 624.954,Z 622.826,A -85,B 0,C 180,E1 30357.232,E2 30357.232} C_VEL
LIN {X 0,Y 624.898,Z 622.826,A -85,B 0,C 180,E1 30354.218,E2 30354.218} C_VEL
LIN {X 0,Y 624.874,Z 622.828,A -85,B 0,C 180,E1 30350.907,E2 30350.907} C_VEL
LIN {X 0,Y 624.934,Z 622.823,A -85,B 0,C 180,E1 30347.988,E2 30347.988} C_VEL
LIN {X 0,Y 624.921,Z 622.821,A -85,B 0,C 180,E1 30344.834,E2 30344.834} C_VEL
LIN {X 0,Y 624.936,Z 622.821,A -85,B 0,C 180,E1 30341.819,E2 30341.819} C_VEL
LIN {X 0,Y 624.946,Z 622.82,A -85,B 0,C 180,E1 30338.614,E2 30338.614} C_VEL
LIN {X 0,Y 624.895,Z 622.825,A -85,B 0,C 180,E1 30335.695,E2 30335.695} C_VEL
LIN {X 0,Y 624.873,Z 622.821,A -85,B 0,C 180,E1 30332.386,E2 30332.386} C_VEL
LIN {X 0,Y 624.947,Z 622.826,A -85,B 0,C 180,E1 30329.451,E2 30329.451} C_VEL
LIN {X 0,Y 624.925,Z 622.815,A -85,B 0,C 180,E1 30326.332,E2 30326.332} C_VEL
LIN {X 0,Y 624.931,Z 622.82,A -85,B 0,C 180,E1 30323.294,E2 30323.294} C_VEL
LIN {X 0,Y 624.942,Z 622.819,A -85,B 0,C 180,E1 30320.144,E2 30320.144} C_VEL
LIN {X 0,Y 624.885,Z 622.82,A -85,B 0,C 180,E1 30317.245,E2 30317.245} C_VEL
LIN {X 0,Y 624.881,Z 622.825,A -85,B 0,C 180,E1 30313.931,E2 30313.931} C_VEL
LIN {X 0,Y 624.945,Z 622.826,A -85,B 0,C 180,E1 30311.001,E2 30311.001} C_VEL
LIN {X 0,Y 624.928,Z 622.821,A -85,B 0,C 180,E1 30307.817,E2 30307.817} C_VEL
LIN {X 0,Y 624.929,Z 622.82,A -85,B 0,C 180,E1 30304.813,E2 30304.813} C_VEL
LIN {X 0,Y 624.939,Z 622.827,A -85,B 0,C 180,E1 30301.63,E2 30301.63} C_VEL
LIN {X 0,Y 624.88,Z 622.827,A -85,B 0,C 180,E1 30298.774,E2 30298.774} C_VEL
LIN {X 0,Y 624.889,Z 622.826,A -85,B 0,C 180,E1 30295.487,E2 30295.487} C_VEL
LIN {X 0,Y 624.946,Z 622.826,A -85,B 0,C 180,E1 30292.516,E2 30292.516} C_VEL
LIN {X 0,Y 624.934,Z 622.821,A -85,B 0,C 180,E1 30289.371,E2 30289.371} C_VEL
LIN {X 0,Y 624.925,Z 622.822,A -85,B 0,C 180,E1 30286.316,E2 30286.316} C_VEL
LIN {X 0,Y 624.932,Z 622.825,A -85,B 0,C 180,E1 30283.15,E2 30283.15} C_VEL
LIN {X 0,Y 624.873,Z 622.866,A -85,B 0,C 180,E1 30280.437,E2 30280.437} C_VEL
LIN {X 0,Y 630.133,Z 643.175,A -85,B 0,C 180,E1 30278.693,E2 30278.693} C_VEL
LIN {X 0,Y 629.493,Z 687.385,A -85,B 0,C 180,E1 30275.375,E2 30275.375} C_VEL
LIN {X 0,Y 628.901,Z 728.568,A -85,B 0,C 180,E1 30272.287,E2 30272.287} C_VEL
LIN {X 0,Y 628.151,Z 771.231,A -85,B 0,C 180,E1 30269.09,E2 30269.09} C_VEL
LIN {X 0,Y 627.462,Z 813.26,A -85,B 0,C 180,E1 30265.937,E2 30265.937} C_VEL
LIN {X 0,Y 627.325,Z 823.819,A -85,B 0,C 180,E1 30265.165,E2 30265.165} C_VEL
LIN {X 0,Y 627.703,Z 831.304,A -85,B 0,C 180,E1 30265.062,E2 30265.062} C_VEL
LIN {X 0,Y 626.802,Z 966.295,A -85,B 0,C 180,E1 30263.399,E2 30263.399} C_VEL
LIN {X 0,Y 626.675,Z 982.505,A -85,B 0,C 180,E1 30263.027,E2 30263.027} C_VEL
LIN {X 0,Y 626.472,Z 998.249,A -85,B 0,C 180,E1 30262.494,E2 30262.494} C_VEL
LIN {X 0,Y 626.201,Z 1012.505,A -85,B 0,C 180,E1 30261.839,E2 30261.839} C_VEL
LIN {X 0,Y 625.893,Z 1027.245,A -85,B 0,C 180,E1 30260.966,E2 30260.966} C_VEL
LIN {X 0,Y 625.553,Z 1040.032,A -85,B 0,C 180,E1 30260,E2 30260} C_VEL
LIN {X 0,Y 625.252,Z 1051.347,A -85,B 0,C 180,E1 30258.941,E2 30258.941} C_VEL
LIN {X 0,Y 624.975,Z 1061.227,A -85,B 0,C 180,E1 30257.79,E2 30257.79} C_VEL
LIN {X 0,Y 624.743,Z 1070.318,A -85,B 0,C 180,E1 30256.454,E2 30256.454} C_VEL
LIN {X 0,Y 624.581,Z 1077.264,A -85,B 0,C 180,E1 30255.124,E2 30255.124} C_VEL
LIN {X 0,Y 624.478,Z 1083.029,A -85,B 0,C 180,E1 30253.611,E2 30253.611} C_VEL
LIN {X 0,Y 624.411,Z 1086.864,A -85,B 0,C 180,E1 30252.013,E2 30252.013} C_VEL
LIN {X 0,Y 624.394,Z 1088.591,A -85,B 0,C 180,E1 30250.515,E2 30250.515} C_VEL
LIN {X 0,Y 624.42,Z 1088.399,A -85,B 0,C 180,E1 30248.934,E2 30248.934} C_VEL
LIN {X 0,Y 624.472,Z 1086.401,A -85,B 0,C 180,E1 30247.45,E2 30247.45} C_VEL
LIN {X 0,Y 624.56,Z 1082.545,A -85,B 0,C 180,E1 30245.971,E2 30245.971} C_VEL
LIN {X 0,Y 624.703,Z 1077.15,A -85,B 0,C 180,E1 30244.588,E2 30244.588} C_VEL
LIN {X 0,Y 624.903,Z 1069.786,A -85,B 0,C 180,E1 30243.208,E2 30243.208} C_VEL
LIN {X 0,Y 625.143,Z 1061.606,A -85,B 0,C 180,E1 30242.015,E2 30242.015} C_VEL
LIN {X 0,Y 625.449,Z 1051.244,A -85,B 0,C 180,E1 30240.822,E2 30240.822} C_VEL
LIN {X 0,Y 625.777,Z 1039.865,A -85,B 0,C 180,E1 30239.769,E2 30239.769} C_VEL
LIN {X 0,Y 626.104,Z 1026.775,A -85,B 0,C 180,E1 30238.808,E2 30238.808} C_VEL
LIN {X 0,Y 626.374,Z 1012.625,A -85,B 0,C 180,E1 30237.985,E2 30237.985} C_VEL
LIN {X 0,Y 626.615,Z 998.038,A -85,B 0,C 180,E1 30237.346,E2 30237.346} C_VEL
LIN {X 0,Y 626.778,Z 984.512,A -85,B 0,C 180,E1 30236.897,E2 30236.897} C_VEL
LIN {X 0,Y 626.87,Z 969.483,A -85,B 0,C 180,E1 30236.537,E2 30236.537} C_VEL
LIN {X 0,Y 627.024,Z 929.201,A -85,B 0,C 180,E1 30236.02,E2 30236.02} C_VEL
LIN {X 0,Y 627.903,Z 826.96,A -85,B 0,C 180,E1 30234.722,E2 30234.722} C_VEL
LIN {X 0,Y 628.514,Z 785.71,A -85,B 0,C 180,E1 30231.674,E2 30231.674} C_VEL
LIN {X 0,Y 628.968,Z 745.787,A -85,B 0,C 180,E1 30228.762,E2 30228.762} C_VEL
LIN {X 0,Y 629.312,Z 704.85,A -85,B 0,C 180,E1 30225.835,E2 30225.835} C_VEL
LIN {X 0,Y 629.289,Z 666.375,A -85,B 0,C 180,E1 30223.142,E2 30223.142} C_VEL
LIN {X 0,Y 629.326,Z 638.627,A -85,B 0,C 180,E1 30221.245,E2 30221.245} C_VEL
LIN {X 0,Y 624.945,Z 622.827,A -85,B 0,C 180,E1 30219.976,E2 30219.976} C_VEL
LIN {X 0,Y 624.934,Z 622.831,A -85,B 0,C 180,E1 30216.919,E2 30216.919} C_VEL
LIN {X 0,Y 624.953,Z 622.823,A -85,B 0,C 180,E1 30213.628,E2 30213.628} C_VEL
LIN {X 0,Y 624.929,Z 622.827,A -85,B 0,C 180,E1 30210.474,E2 30210.474} C_VEL
LIN {X 0,Y 624.944,Z 622.827,A -85,B 0,C 180,E1 30207.37,E2 30207.37} C_VEL
LIN {X 0,Y 624.928,Z 622.825,A -85,B 0,C 180,E1 30204.266,E2 30204.266} C_VEL
LIN {X 0,Y 624.942,Z 622.824,A -85,B 0,C 180,E1 30200.891,E2 30200.891} C_VEL
LIN {X 0,Y 624.949,Z 622.826,A -85,B 0,C 180,E1 30197.778,E2 30197.778} C_VEL
LIN {X 0,Y 624.921,Z 622.823,A -85,B 0,C 180,E1 30194.6,E2 30194.6} C_VEL
LIN {X 0,Y 624.933,Z 622.824,A -85,B 0,C 180,E1 30191.603,E2 30191.603} C_VEL
LIN {X 0,Y 624.94,Z 622.825,A -85,B 0,C 180,E1 30188.371,E2 30188.371} C_VEL
LIN {X 0,Y 624.949,Z 622.89,A -85,B 0,C 180,E1 30186.564,E2 30186.564} C_VEL
LIN {X 0,Y 633.074,Z 648.444,A -85,B 0,C 180,E1 30183.739,E2 30183.739} C_VEL
LIN {X 0,Y 634.621,Z 654.207,A -85,B 0,C 180,E1 30183.14,E2 30183.14} C_VEL
LIN {X 0,Y 633.339,Z 681.104,A -85,B 0,C 180,E1 30180.868,E2 30180.868} C_VEL
LIN {X 0,Y 638.777,Z 708.09,A -85,B 0,C 180,E1 30180.204,E2 30180.204} C_VEL
LIN {X 0,Y 636.006,Z 907.215,A -85,B 0,C 180,E1 30177.706,E2 30177.706} C_VEL
LIN {X 0,Y 634.949,Z 986.607,A -85,B 0,C 180,E1 30176.703,E2 30176.703} C_VEL
LIN {X 0,Y 634.263,Z 1008.744,A -85,B 0,C 180,E1 30176.258,E2 30176.258} C_VEL
LIN {X 0,Y 633.453,Z 1030.601,A -85,B 0,C 180,E1 30175.652,E2 30175.652} C_VEL
LIN {X 0,Y 632.526,Z 1051.448,A -85,B 0,C 180,E1 30174.914,E2 30174.914} C_VEL
LIN {X 0,Y 631.492,Z 1072.017,A -85,B 0,C 180,E1 30174.01,E2 30174.01} C_VEL
LIN {X 0,Y 630.406,Z 1091.672,A -85,B 0,C 180,E1 30172.964,E2 30172.964} C_VEL
LIN {X 0,Y 629.281,Z 1111.271,A -85,B 0,C 180,E1 30171.728,E2 30171.728} C_VEL
LIN {X 0,Y 628.255,Z 1128.666,A -85,B 0,C 180,E1 30170.445,E2 30170.445} C_VEL
LIN {X 0,Y 627.311,Z 1144.742,A -85,B 0,C 180,E1 30169.054,E2 30169.054} C_VEL
LIN {X 0,Y 626.414,Z 1160.607,A -85,B 0,C 180,E1 30167.461,E2 30167.461} C_VEL
LIN {X 0,Y 625.689,Z 1174.534,A -85,B 0,C 180,E1 30165.836,E2 30165.836} C_VEL
LIN {X 0,Y 625.091,Z 1186.726,A -85,B 0,C 180,E1 30164.165,E2 30164.165} C_VEL
LIN {X 0,Y 624.634,Z 1197.734,A -85,B 0,C 180,E1 30162.385,E2 30162.385} C_VEL
LIN {X 0,Y 624.343,Z 1206.431,A -85,B 0,C 180,E1 30160.705,E2 30160.705} C_VEL
LIN {X 0,Y 624.107,Z 1214.531,A -85,B 0,C 180,E1 30158.753,E2 30158.753} C_VEL
LIN {X 0,Y 623.971,Z 1221.149,A -85,B 0,C 180,E1 30156.716,E2 30156.716} C_VEL
LIN {X 0,Y 623.92,Z 1225.824,A -85,B 0,C 180,E1 30154.779,E2 30154.779} C_VEL
LIN {X 0,Y 623.908,Z 1228.787,A -85,B 0,C 180,E1 30152.846,E2 30152.846} C_VEL
LIN {X 0,Y 623.907,Z 1230.326,A -85,B 0,C 180,E1 30150.733,E2 30150.733} C_VEL
LIN {X 0,Y 623.901,Z 1230.208,A -85,B 0,C 180,E1 30148.805,E2 30148.805} C_VEL
LIN {X 0,Y 623.902,Z 1228.439,A -85,B 0,C 180,E1 30146.875,E2 30146.875} C_VEL
LIN {X 0,Y 623.926,Z 1225.011,A -85,B 0,C 180,E1 30144.85,E2 30144.85} C_VEL
LIN {X 0,Y 623.993,Z 1220.125,A -85,B 0,C 180,E1 30142.911,E2 30142.911} C_VEL
LIN {X 0,Y 624.133,Z 1213.46,A -85,B 0,C 180,E1 30140.966,E2 30140.966} C_VEL
LIN {X 0,Y 624.388,Z 1204.579,A -85,B 0,C 180,E1 30138.92,E2 30138.92} C_VEL
LIN {X 0,Y 624.707,Z 1196.122,A -85,B 0,C 180,E1 30137.332,E2 30137.332} C_VEL
LIN {X 0,Y 625.179,Z 1184.642,A -85,B 0,C 180,E1 30135.551,E2 30135.551} C_VEL
LIN {X 0,Y 625.785,Z 1171.784,A -85,B 0,C 180,E1 30133.857,E2 30133.857} C_VEL
LIN {X 0,Y 626.522,Z 1157.476,A -85,B 0,C 180,E1 30132.251,E2 30132.251} C_VEL
LIN {X 0,Y 627.372,Z 1141.642,A -85,B 0,C 180,E1 30130.736,E2 30130.736} C_VEL
LIN {X 0,Y 628.362,Z 1123.635,A -85,B 0,C 180,E1 30129.263,E2 30129.263} C_VEL
LIN {X 0,Y 629.342,Z 1105.172,A -85,B 0,C 180,E1 30127.978,E2 30127.978} C_VEL
LIN {X 0,Y 630.368,Z 1085.722,A -85,B 0,C 180,E1 30126.834,E2 30126.834} C_VEL
LIN {X 0,Y 631.314,Z 1065.669,A -85,B 0,C 180,E1 30125.848,E2 30125.848} C_VEL
LIN {X 0,Y 632.269,Z 1043.58,A -85,B 0,C 180,E1 30124.956,E2 30124.956} C_VEL
LIN {X 0,Y 633.109,Z 1022.022,A -85,B 0,C 180,E1 30124.262,E2 30124.262} C_VEL
LIN {X 0,Y 633.773,Z 1000.3,A -85,B 0,C 180,E1 30123.733,E2 30123.733} C_VEL
LIN {X 0,Y 634.303,Z 977.589,A -85,B 0,C 180,E1 30123.345,E2 30123.345} C_VEL
LIN {X 0,Y 636.194,Z 825.052,A -85,B 0,C 180,E1 30121.428,E2 30121.428} C_VEL
LIN {X 0,Y 638.622,Z 707.033,A -85,B 0,C 180,E1 30119.806,E2 30119.806} C_VEL
LIN {X 0,Y 632.789,Z 676.249,A -85,B 0,C 180,E1 30118.957,E2 30118.957} C_VEL
LIN {X 0,Y 633.967,Z 652.442,A -85,B 0,C 180,E1 30116.878,E2 30116.878} C_VEL
LIN {X 0,Y 629.77,Z 637.209,A -85,B 0,C 180,E1 30115.139,E2 30115.139} C_VEL
LIN {X 0,Y 625.837,Z 625.664,A -85,B 0,C 180,E1 30113.634,E2 30113.634} C_VEL
LIN {X 0,Y 624.935,Z 622.827,A -85,B 0,C 180,E1 30113.244,E2 30113.244} C_VEL
LIN {X 0,Y 624.938,Z 622.825,A -85,B 0,C 180,E1 30109.969,E2 30109.969} C_VEL
LIN {X 0,Y 624.949,Z 622.823,A -85,B 0,C 180,E1 30106.781,E2 30106.781} C_VEL
LIN {X 0,Y 624.916,Z 622.828,A -85,B 0,C 180,E1 30103.601,E2 30103.601} C_VEL
LIN {X 0,Y 624.957,Z 622.823,A -85,B 0,C 180,E1 30100.511,E2 30100.511} C_VEL
LIN {X 0,Y 624.903,Z 622.828,A -85,B 0,C 180,E1 30097.449,E2 30097.449} C_VEL
LIN {X 0,Y 624.951,Z 622.825,A -85,B 0,C 180,E1 30094.389,E2 30094.389} C_VEL
LIN {X 0,Y 624.922,Z 622.884,A -85,B 0,C 180,E1 30092.74,E2 30092.74} C_VEL
LIN {X 0,Y 628.123,Z 632.496,A -85,B 0,C 180,E1 30091.258,E2 30091.258} C_VEL
LIN {X 0,Y 635.371,Z 645.5,A -85,B 0,C 180,E1 30090.553,E2 30090.553} C_VEL
LIN {X 0,Y 639.316,Z 653.728,A -85,B 0,C 180,E1 30090.186,E2 30090.186} C_VEL
LIN {X 0,Y 636.609,Z 774.784,A -85,B 0,C 180,E1 30088.497,E2 30088.497} C_VEL
LIN {X 0,Y 634.69,Z 914.337,A -85,B 0,C 180,E1 30086.728,E2 30086.728} C_VEL
LIN {X 0,Y 634.271,Z 938.071,A -85,B 0,C 180,E1 30086.371,E2 30086.371} C_VEL
LIN {X 0,Y 633.68,Z 961.14,A -85,B 0,C 180,E1 30085.853,E2 30085.853} C_VEL
LIN {X 0,Y 632.953,Z 982.084,A -85,B 0,C 180,E1 30085.224,E2 30085.224} C_VEL
LIN {X 0,Y 632.103,Z 1002.49,A -85,B 0,C 180,E1 30084.438,E2 30084.438} C_VEL
LIN {X 0,Y 631.16,Z 1021.792,A -85,B 0,C 180,E1 30083.531,E2 30083.531} C_VEL
LIN {X 0,Y 630.189,Z 1040.529,A -85,B 0,C 180,E1 30082.483,E2 30082.483} C_VEL
LIN {X 0,Y 629.106,Z 1059.061,A -85,B 0,C 180,E1 30081.248,E2 30081.248} C_VEL
LIN {X 0,Y 628.095,Z 1075.921,A -85,B 0,C 180,E1 30079.92,E2 30079.92} C_VEL
LIN {X 0,Y 627.096,Z 1092.362,A -85,B 0,C 180,E1 30078.405,E2 30078.405} C_VEL
LIN {X 0,Y 626.224,Z 1107.174,A -85,B 0,C 180,E1 30076.8,E2 30076.8} C_VEL
LIN {X 0,Y 625.485,Z 1120.656,A -85,B 0,C 180,E1 30075.083,E2 30075.083} C_VEL
LIN {X 0,Y 624.898,Z 1132.227,A -85,B 0,C 180,E1 30073.323,E2 30073.323} C_VEL
LIN {X 0,Y 624.461,Z 1142.516,A -85,B 0,C 180,E1 30071.454,E2 30071.454} C_VEL
LIN {X 0,Y 624.19,Z 1151.481,A -85,B 0,C 180,E1 30069.499,E2 30069.499} C_VEL
LIN {X 0,Y 624.034,Z 1158.225,A -85,B 0,C 180,E1 30067.644,E2 30067.644} C_VEL
LIN {X 0,Y 623.948,Z 1163.869,A -85,B 0,C 180,E1 30065.612,E2 30065.612} C_VEL
LIN {X 0,Y 623.915,Z 1167.663,A -85,B 0,C 180,E1 30063.677,E2 30063.677} C_VEL
